	IF arrAxisCtrl[P3AxisNo.P3M1_ColdpreWhirling].Cmd.arrbRealPoint[1] AND NOT arrAxisCtrl[P3AxisNo.P3M1_ColdpreWhirling].Status.Moving THEN
		ColdpreWhirlTorMark:=FALSE;//冷压上料夹旋转力矩超限报警标志
		Init_step[1]:=170;
	END_IF	
	

	
	
170://冷压上料夹旋转在初始位且已停止，则冷压上料夹升降开始回零
INIT_TON[7].IN:=TRUE;
IF arrAxisCtrl[P3AxisNo.P3M1_ColdpreWhirling].Cmd.arrbRealPoint[1] AND NOT arrAxisCtrl[P3AxisNo.P3M1_ColdpreWhirling].Status.Moving AND  INIT_TON[7].Q THEN
	arrAxisCtrl[P3AxisNo.P3M1_ColdpreUpDown].Cmd.bHome:=TRUE;//冷压上料升降回零
	INIT_TON[7].IN:=FALSE;
	Init_step[1]:=180;
	END_IF
	

180://冷压上料夹升降回零完成
INIT_TON[9].IN:=TRUE;
	IF  arrAxisCtrl[P3AxisNo.P3M1_ColdpreUpDown].Status.Homed AND NOT arrAxisCtrl[P3AxisNo.P3M1_ColdpreUpDown].Status.Moving  AND  INIT_TON[9].Q  THEN
		Init_step[1]:=190;
		arrAxisCtrl[P3AxisNo.P3M1_ColdpreUpDown].Cmd.bHome:=FALSE;	
		INIT_TON[9].IN:=FALSE;
	END_IF

190://冷压上料夹升降到初始位
	IF  NOT arrAxisCtrl[P3AxisNo.P3M1_ColdpreUpDown].Cmd.arrbRealPoint[1] 
	AND NOT arrAxisCtrl[P3AxisNo.P3M1_ColdpreUpDown].Status.Error 
	AND arrAxisCtrl[P3AxisNo.P3M1_ColdpreUpDown].Status.Homed 
	AND arrAxisCtrl[P3AxisNo.P3M1_ColdpreUpDown].Status.Enabled 
	AND arrAxisCtrl[P3AxisNo.P3M1_ColdpreUpDown].Status.NoMoving THEN
		arrAxisCtrl[P3AxisNo.P3M1_ColdpreUpDown].Cmd.iGoSetPos:=1;	//冷压上料升降回初始位
	END_IF

	
	IF  arrAxisCtrl[P3AxisNo.P3M1_ColdpreUpDown].Cmd.arrbRealPoint[1] AND NOT arrAxisCtrl[P3AxisNo.P3M1_ColdpreUpDown].Status.Moving  THEN
		Init_step[1]:=200;
	END_IF


	
200:
Step30:=1;
Init_step[1]:=999;

999://冷压上料初始化完成
IF Init_step[1]=999 THEN
INIT_TON[20].IN:=FALSE;
LateBlanking_init_OK[1]:=TRUE;
END_IF

END_CASE
END_IF


IF 	arrAxisCtrl[P3AxisNo.P3M1_ColdpreLine].Status.Error OR arrAxisCtrl[P3AxisNo.P3M1_ColdpreUpDown].Status.Error OR
	arrAxisCtrl[P3AxisNo.P3M1_ColdpreWhirling].Status.Error OR  arrAxisCtrl[P3AxisNo.P3M1_ColdpreRetracting].Status.Error THEN
	Init_step[1]:=0;
END_IF

IF   P3_SystemRUN.btnStop OR NOT P3Button.LateStop THEN
	Init_step[1]:=0;
	Init_step[2]:=0;
	Init_step[3]:=0;
	Init_step[4]:=0;
	Init_step[5]:=0;
	Init_step[6]:=0;
	Init_step[7]:=0;
	Init_step[8]:=0;
END_IF

END_PROGRAM

// ---- P3POUs/POUs/Init/L_Init2.TcPOU
PROGRAM L_Init2
VAR
	INIT_TON  :ARRAY[1..20] OF Tc2_Standard.TON;
END_VAR

INIT_TON[1](PT:=T#2S);
INIT_TON[2](PT:=T#2S);
INIT_TON[3](PT:=T#2S);
INIT_TON[4](PT:=T#2S);
INIT_TON[5](PT:=T#2S);
INIT_TON[6](PT:=T#2S);
INIT_TON[7](PT:=T#2S);
INIT_TON[8](PT:=T#2S);
INIT_TON[9](PT:=T#2S);
INIT_TON[10](PT:=T#3S);
INIT_TON[20](PT:=T#60S);//冷压驱动回原超时计时

IF INIT_TON[20].Q THEN
	Init_step[2]:=0;
	P3_Error[121]:=TRUE;//冷压驱动回原超时报警
	INIT_TON[20].IN:=FALSE;
END_IF
//冷压托板开合回原条件
IF arrAxisCtrl[P3AxisNo.P3M1_ColdpreSupPlateLine].Status.Enabled AND NOT arrAxisCtrl[P3AxisNo.P3M1_ColdpreSupPlateLine].Status.Error AND P3_SystemRUN.iMode=3 
AND (arrAxisCtrlV2[P3AxisNo.P3_M2_OvenRetracting].Cmd.arrbRealPoint[43] OR (LREAL_TO_REAL(arrAxisCtrlV2[P3AxisNo.P3_M2_OvenCarrying].Status.fActPos)>=(arrAxisParV2[P3AxisNo.P3_M2_OvenCarrying].arrTargetPoint[1]-5)
AND  arrAxisCtrlV2[P3AxisNo.P3_M2_OvenCarrying].Status.Homed)) 
AND (arrAxisCtrl[P3AxisNo.P3M1_ColdpreRetracting].Cmd.arrbRealPoint[1] OR (LREAL_TO_REAL(arrAxisCtrl[P3AxisNo.P3M1_ColdpreLine].Status.fActPos)<=(arrAxisPar[P3AxisNo.P3M1_ColdpreLine].arrTargetPoint[2]+5)
AND  arrAxisCtrl[P3AxisNo.P3M1_ColdpreLine].Status.Homed))
AND  arrAxisCtrl[P3AxisNo.P3M1_ColdpreActuated].Cmd.arrbRealPoint[1]  THEN
   arrAxisCtrl[P3AxisNo.P3M1_ColdpreSupPlateLine].Cmd.Home_Condition:=TRUE;
   ELSE 
   arrAxisCtrl[P3AxisNo.P3M1_ColdpreSupPlateLine].Cmd.Home_Condition:=FALSE;
 END_IF

//冷压驱动回原条件
IF arrAxisCtrl[P3AxisNo.P3M1_ColdpreActuated].Status.Enabled AND NOT arrAxisCtrl[P3AxisNo.P3M1_ColdpreActuated].Status.Error AND P3_SystemRUN.iMode=3 THEN
   arrAxisCtrl[P3AxisNo.P3M1_ColdpreActuated].Cmd.Home_Condition:=TRUE;
   ELSE 
   arrAxisCtrl[P3AxisNo.P3M1_ColdpreActuated].Cmd.Home_Condition:=FALSE;
 END_IF










///////////////////////冷压初始化
IF P3_SystemRUN.iMode=3  THEN
IF LateBlanking_init_start[2]  THEN
	Init_step[2]:=1;
	LateBlanking_init_OK[2]:=FALSE;
	LateBlanking_init_start[2]:=FALSE;
END_IF
END_IF


IF P3_SystemRUN.iMode=3 AND LateBlanking_init_OK[1] AND  LateBlanking_init_OK[3] THEN
CASE Init_step[2] OF
1://冷压电芯记忆清除
	INIT_TON[20].IN:=TRUE;
	Permit_Cold_Press:=FALSE;	
	Cold_Press_Finish:=FALSE;	
	Step31:=0;
	INIT_TON[10].IN:=FALSE;
	ColdPress_start:=FALSE;
	MEMSET(ADR(CellMemory[CellNo.Coldpress]),0,SIZEOF(CellMemory[CellNo.Coldpress]));
	Init_step[2]:=10;//信号复位
	
10://冷压麦拉张紧气缸打开
arrCyCtrl[P3CYNo.P3ColdPressTensed].Cmd.bON:=TRUE;
Init_step[2]:=20;//气缸打开

20://冷压驱动停止信号复位
	arrAxisCtrl[P3AxisNo.P3M1_ColdpreActuated].Cmd.bStop:=TRUE;
	arrAxisCtrl[P3AxisNo.P3M1_ColdpreSupPlateLine].Cmd.bStop:=TRUE;//轴停止
	INIT_TON[1].IN:=TRUE;
	IF INIT_TON[1].Q THEN
		Init_step[2]:=30;
	arrAxisCtrl[P3AxisNo.P3M1_ColdpreActuated].Cmd.bStop:=FALSE;
	arrAxisCtrl[P3AxisNo.P3M1_ColdpreSupPlateLine].Cmd.bStop:=FALSE;
	INIT_TON[1].IN:=FALSE;	
	END_IF

30://冷压驱动轴复位
    arrAxisCtrl[P3AxisNo.P3M1_ColdpreActuated].Cmd.bReset:=TRUE;
	arrAxisCtrl[P3AxisNo.P3M1_ColdpreSupPlateLine].Cmd.bReset:=TRUE;//轴复位
	INIT_TON[2].IN:=TRUE;
	
	IF INIT_TON[2].Q THEN
		Init_step[2]:=40;
	    arrAxisCtrl[P3AxisNo.P3M1_ColdpreActuated].Cmd.bReset:=FALSE;
		arrAxisCtrl[P3AxisNo.P3M1_ColdpreSupPlateLine].Cmd.bReset:=FALSE;
		INIT_TON[2].IN:=FALSE;
	END_IF

40://冷压驱动、冷压托板开合轴上使能
    arrAxisCtrl[P3AxisNo.P3M1_ColdpreActuated].Cmd.bEnable:=TRUE;
	arrAxisCtrl[P3AxisNo.P3M1_ColdpreSupPlateLine].Cmd.bEnable:=TRUE;//轴上使能
	IF arrAxisCtrl[P3AxisNo.P3M1_ColdpreActuated].Status.Enabled AND arrAxisCtrl[P3AxisNo.P3M1_ColdpreSupPlateLine].Status.Enabled THEN
		Init_step[2]:=50;
	END_IF

50://冷压驱动开始回零
arrAxisCtrl[P3AxisNo.P3M1_ColdpreActuated].Cmd.bHome:=TRUE;
Init_step[2]:=60;

60://冷压驱动回零完成
INIT_TON[3].IN:=TRUE;
IF arrAxisCtrl[P3AxisNo.P3M1_ColdpreActuated].Status.Homed AND NOT arrAxisCtrl[P3AxisNo.P3M1_ColdpreActuated].Status.Moving AND INIT_TON[3].Q THEN
	Init_step[2]:=70;
    arrAxisCtrl[P3AxisNo.P3M1_ColdpreActuated].Cmd.bHome:=FALSE;
	INIT_TON[3].IN:=FALSE;
END_IF

70://冷压驱动到初始位
IF NOT arrAxisCtrl[P3AxisNo.P3M1_ColdpreActuated].Cmd.arrbRealPoint[1] AND NOT arrAxisCtrl[P3AxisNo.P3M1_ColdpreActuated].Status.Error AND arrAxisCtrl[P3AxisNo.P3M1_ColdpreActuated].Status.Homed 
	AND arrAxisCtrl[P3AxisNo.P3M1_ColdpreActuated].Status.Enabled AND arrAxisCtrl[P3AxisNo.P3M1_ColdpreActuated].Status.NoMoving THEN
	arrAxisCtrl[P3AxisNo.P3M1_ColdpreActuated].Cmd.iGoSetPos:=1;//冷压驱动回初始位	
END_IF

IF 	arrAxisCtrl[P3AxisNo.P3M1_ColdpreActuated].Cmd.arrbRealPoint[1]  AND NOT arrAxisCtrl[P3AxisNo.P3M1_ColdpreActuated].Status.Moving THEN
	Init_step[2]:=80;
END_IF


80://冷压托板开合开始回零
arrAxisCtrl[P3AxisNo.P3M1_ColdpreSupPlateLine].Cmd.bHome:=TRUE;
Init_step[2]:=90;
	
90://冷压托板开合回零完成，冷压麦拉张紧气缸打开
INIT_TON[8].IN:=TRUE;
	IF 	arrAxisCtrl[P3AxisNo.P3M1_ColdpreSupPlateLine].Status.Homed AND arrAxisCtrl[P3AxisNo.P3M1_ColdpreSupPlateLine].Status.NoMoving AND  INIT_TON[8].Q THEN
		Init_step[2]:=100;
		arrAxisCtrl[P3AxisNo.P3M1_ColdpreSupPlateLine].Cmd.bHome:=FALSE;
		arrCyCtrl[P3CYNo.P3ColdPressTensed].Cmd.bON:=TRUE;//冷压麦拉膜气缸张紧
		INIT_TON[8].IN:=FALSE;
		END_IF
100://冷压托板开合到张开位检查有无电芯
    IF  NOT arrAxisCtrl[P3AxisNo.P3M1_ColdpreSupPlateLine].Cmd.arrbRealPoint[2] AND NOT arrAxisCtrl[P3AxisNo.P3M1_ColdpreSupPlateLine].Status.Error AND arrAxisCtrl[P3AxisNo.P3M1_ColdpreSupPlateLine].Status.Homed 
		AND arrAxisCtrl[P3AxisNo.P3M1_ColdpreSupPlateLine].Status.Enabled AND arrAxisCtrl[P3AxisNo.P3M1_ColdpreSupPlateLine].Status.NoMoving THEN
		arrAxisCtrl[P3AxisNo.P3M1_ColdpreSupPlateLine].Cmd.iGoSetPos:=2;//冷压托板开合去张开位
	END_IF 
    IF arrAxisCtrl[P3AxisNo.P3M1_ColdpreSupPlateLine].Cmd.arrbRealPoint[2] 
	AND arrAxisCtrl[P3AxisNo.P3M1_ColdpreSupPlateLine].Status.NoMoving 
	AND NOT P3Senser.P3_ColdEmptyPress THEN
		Init_step[2]:=110;	
	ELSIF arrAxisCtrl[P3AxisNo.P3M1_ColdpreSupPlateLine].Cmd.arrbRealPoint[2] 
	AND arrAxisCtrl[P3AxisNo.P3M1_ColdpreSupPlateLine].Status.NoMoving 
	AND  P3Senser.P3_ColdEmptyPress THEN
		Init_step[2]:=888;	
		P3_Error[74]:=TRUE;//冷压初始化时，电芯未取走报警！
	END_IF
	
110://冷压托板开合到初始位
	IF  NOT arrAxisCtrl[P3AxisNo.P3M1_ColdpreSupPlateLine].Cmd.arrbRealPoint[1] AND NOT arrAxisCtrl[P3AxisNo.P3M1_ColdpreSupPlateLine].Status.Error AND arrAxisCtrl[P3AxisNo.P3M1_ColdpreSupPlateLine].Status.Homed 
		AND arrAxisCtrl[P3AxisNo.P3M1_ColdpreSupPlateLine].Status.Enabled AND arrAxisCtrl[P3AxisNo.P3M1_ColdpreSupPlateLine].Status.NoMoving THEN
		arrAxisCtrl[P3AxisNo.P3M1_ColdpreSupPlateLine].Cmd.iGoSetPos:=1;//冷压托板开合回初始位	
	END_IF
    IF  arrAxisCtrl[P3AxisNo.P3M1_ColdpreSupPlateLine].Cmd.arrbRealPoint[1] AND arrAxisCtrl[P3AxisNo.P3M1_ColdpreSupPlateLine].Status.NoMoving THEN
		Init_step[2]:=120;
		
	END_IF

	
120:
Step31:=1;
Init_step[2]:=999;

999://冷压回零完成
IF Init_step[2]=999 THEN
INIT_TON[20].IN:=FALSE;
LateBlanking_init_OK[2]:=TRUE;
END_IF

END_CASE
END_IF

IF arrAxisCtrl[P3AxisNo.P3M1_ColdpreSupPlateLine].Status.Error OR arrAxisCtrl[P3AxisNo.P3M1_ColdpreActuated].Status.Error THEN
	Init_step[2]:=0;
END_IF

END_PROGRAM

// ---- P3POUs/POUs/Init/L_Init3.TcPOU
PROGRAM L_Init3
VAR
	INIT_TON  :ARRAY[1..20] OF Tc2_Standard.TON;
END_VAR

INIT_TON[1](PT:=T#2S);
INIT_TON[2](PT:=T#2S);
INIT_TON[3](PT:=T#2S);
INIT_TON[4](PT:=T#2S);
INIT_TON[5](PT:=T#2S);
INIT_TON[6](PT:=T#2S);
INIT_TON[7](PT:=T#2S);
INIT_TON[8](PT:=T#2S);
INIT_TON[9](PT:=T#2S);
INIT_TON[10](PT:=T#3S);
INIT_TON[20](PT:=T#90S);//烤箱上料回原超时计时

IF INIT_TON[20].Q THEN
	Init_step[3]:=0;
	P3_Error[122]:=TRUE;//烤箱上料回原超时报警
	INIT_TON[20].IN:=FALSE;
END_IF
//烤箱上料夹搬运回原条件
IF arrAxisCtrlV2[P3AxisNo.P3_M2_OvenCarrying].Status.Enabled AND NOT arrAxisCtrlV2[P3AxisNo.P3_M2_OvenCarrying].Status.Error AND P3_SystemRUN.iMode=3 
AND arrAxisCtrlV2[P3AxisNo.P3_M2_OvenRetracting].Cmd.arrbRealPoint[43] AND Oven_CYOFF_condition THEN
   arrAxisCtrlV2[P3AxisNo.P3_M2_OvenCarrying].Cmd.Home_Condition:=TRUE;
   ELSE 
   arrAxisCtrlV2[P3AxisNo.P3_M2_OvenCarrying].Cmd.Home_Condition:=FALSE;
 END_IF

//烤箱上料夹进退回原条件
IF arrAxisCtrlV2[P3AxisNo.P3_M2_OvenRetracting].Status.Enabled AND NOT arrAxisCtrl[P3AxisNo.P3_M2_OvenRetracting].Status.Error AND P3_SystemRUN.iMode=3  THEN
   arrAxisCtrlV2[P3AxisNo.P3_M2_OvenRetracting].Cmd.Home_Condition:=TRUE;
   ELSE 
   arrAxisCtrlV2[P3AxisNo.P3_M2_OvenRetracting].Cmd.Home_Condition:=FALSE;
 END_IF

//烤箱上料夹升降回原条件
IF arrAxisCtrlV2[P3AxisNo.P3_M2_OvenUpDown].Status.Enabled AND NOT arrAxisCtrlV2[P3AxisNo.P3_M2_OvenUpDown].Status.Error AND P3_SystemRUN.iMode=3  
AND arrAxisCtrlV2[P3AxisNo.P3_M2_OvenRetracting].Cmd.arrbRealPoint[43] AND Oven_CYOFF_condition THEN
   arrAxisCtrlV2[P3AxisNo.P3_M2_OvenUpDown].Cmd.Home_Condition:=TRUE;
   ELSE 
   arrAxisCtrlV2[P3AxisNo.P3_M2_OvenUpDown].Cmd.Home_Condition:=FALSE;
 END_IF





//烤箱上下料初始化
IF P3_SystemRUN.iMode=3 THEN
IF LateBlanking_init_start[3] AND Oven_CYOFF_condition THEN
	Init_step[3]:=1;
	LateBlanking_init_OK[3]:=FALSE;
	LateBlanking_init_start[3]:=FALSE;
	ELSIF LateBlanking_init_start[3] AND NOT Oven_CYOFF_condition THEN
		Init_step[3]:=0;
		LateBlanking_init_OK[3]:=FALSE;
		LateBlanking_init_start[3]:=FALSE;
		P3_Error[28]:=TRUE;//初始化过程中，烤箱门未完成关闭，请完全关闭再重新启动烤箱初始化
END_IF
END_IF



IF P3_SystemRUN.iMode=3 THEN
CASE Init_step[3] OF

1:	//冷压下料到烤箱及烤箱下料到热压时电芯记忆清除
	INIT_TON[20].IN:=TRUE;
	Step32:=0;	
	INIT_TON[10].IN:=FALSE;
	MEMSET(ADR(CellMemory[CellNo.OvenMoveClip1]),0,SIZEOF(CellMemory[CellNo.OvenMoveClip1]));
	MEMSET(ADR(CellMemory[CellNo.OvenMoveClip2]),0,SIZEOF(CellMemory[CellNo.OvenMoveClip2]));
	Init_step[3]:=10;//信号复位
	
10://烤箱上料夹气缸关闭
arrCyCtrl[P3CYNo.P3OvenMoveClip].Cmd.bOFF:=TRUE;
IF  arrCyCtrl[P3CYNo.P3OvenMoveClip].Status.OFFState AND NOT arrCyCtrl[P3CYNo.P3OvenMoveClip].Status.Error2  THEN
	Init_step[3]:=20;
END_IF//



20://烤箱上料夹各轴停止信号复位
	arrAxisCtrlV2[P3AxisNo.P3_M2_OvenCarrying].Cmd.bStop:=TRUE;       arrAxisCtrlV2[P3AxisNo.P3_M2_OvenUpDown].Cmd.bStop:=TRUE;
	arrAxisCtrlV2[P3AxisNo.P3_M2_OvenRetracting].Cmd.bStop:=TRUE;     //轴停止
	INIT_TON[1].IN:=TRUE;
	IF INIT_TON[1].Q THEN
		Init_step[3]:=30;
		arrAxisCtrlV2[P3AxisNo.P3_M2_OvenCarrying].Cmd.bStop:=FALSE;       arrAxisCtrlV2[P3AxisNo.P3_M2_OvenUpDown].Cmd.bStop:=FALSE;
		arrAxisCtrlV2[P3AxisNo.P3_M2_OvenRetracting].Cmd.bStop:=FALSE;    
		INIT_TON[1].IN:=FALSE;	
	END_IF

30://烤箱上料夹各轴复位
	arrAxisCtrlV2[P3AxisNo.P3_M2_OvenCarrying].Cmd.bReset:=TRUE;       arrAxisCtrlV2[P3AxisNo.P3_M2_OvenUpDown].Cmd.bReset:=TRUE;
	arrAxisCtrlV2[P3AxisNo.P3_M2_OvenRetracting].Cmd.bReset:=TRUE;     //轴复位
	INIT_TON[2].IN:=TRUE;
	
	IF INIT_TON[2].Q THEN
		Init_step[3]:=40;
		arrAxisCtrlV2[P3AxisNo.P3_M2_OvenCarrying].Cmd.bReset:=FALSE;       arrAxisCtrlV2[P3AxisNo.P3_M2_OvenUpDown].Cmd.bReset:=FALSE;
		arrAxisCtrlV2[P3AxisNo.P3_M2_OvenRetracting].Cmd.bReset:=FALSE;     
		INIT_TON[2].IN:=FALSE;
	END_IF

40://烤箱上料夹各轴上使能
	arrAxisCtrlV2[P3AxisNo.P3_M2_OvenCarrying].Cmd.bEnable:=TRUE;       arrAxisCtrlV2[P3AxisNo.P3_M2_OvenUpDown].Cmd.bEnable:=TRUE;
	arrAxisCtrlV2[P3AxisNo.P3_M2_OvenRetracting].Cmd.bEnable:=TRUE;     //轴上使能
	IF  arrAxisCtrlV2[P3AxisNo.P3_M2_OvenCarrying].Status.Enabled AND arrAxisCtrlV2[P3AxisNo.P3_M2_OvenUpDown].Status.Enabled
		AND arrAxisCtrlV2[P3AxisNo.P3_M2_OvenRetracting].Status.Enabled  THEN
		Init_step[3]:=50;
	END_IF

50://烤箱上料夹进退开始回零
arrAxisCtrlV2[P3AxisNo.P3_M2_OvenRetracting].Cmd.bHome:=TRUE;//烤箱上料进退回零
Init_step[3]:=60;

60://烤箱上料夹进退回零完成
INIT_TON[4].IN:=TRUE;
IF arrAxisCtrlV2[P3AxisNo.P3_M2_OvenRetracting].Status.Homed AND NOT arrAxisCtrlV2[P3AxisNo.P3_M2_OvenRetracting].Status.Moving AND  INIT_TON[4].Q  THEN
	Init_step[3]:=70;
    arrAxisCtrlV2[P3AxisNo.P3_M2_OvenRetracting].Cmd.bHome:=FALSE;
	INIT_TON[4].IN:=FALSE;
END_IF

70://烤箱上料夹进退到初始位
IF  NOT arrAxisCtrlV2[P3AxisNo.P3_M2_OvenRetracting].Cmd.arrbRealPoint[43] AND NOT arrAxisCtrlV2[P3AxisNo.P3_M2_OvenRetracting].Status.Error AND arrAxisCtrlV2[P3AxisNo.P3_M2_OvenRetracting].Status.Homed 
	AND arrAxisCtrlV2[P3AxisNo.P3_M2_OvenRetracting].Status.Enabled AND arrAxisCtrlV2[P3AxisNo.P3_M2_OvenRetracting].Status.NoMoving THEN
	arrAxisCtrlV2[P3AxisNo.P3_M2_OvenRetracting].Cmd.iGoSetPos:=43;
	OvenRetractTorMark:=TRUE;//烤箱上料夹进退力矩超限报警标志
END_IF 

IF  arrAxisCtrlV2[P3AxisNo.P3_M2_OvenRetracting].Cmd.arrbRealPoint[43]  AND Oven_POS1  AND NOT arrAxisCtrlV2[P3AxisNo.P3_M2_OvenRetracting].Status.Moving THEN
	OvenRetractTorMark:=FALSE;//烤箱上料夹进退力矩超限报警标志
	Init_step[3]:=90;
	
END_IF



90://没有烤箱气缸报警或轴急停且烤箱全部关闭，则烤箱上料夹升降开始回零
	IF  NOT Oven_CY_STOP AND Oven_CYOFF_condition THEN
		arrAxisCtrlV2[P3AxisNo.P3_M2_OvenUpDown].Cmd.bHome:=TRUE;//烤箱上料升降回零
		Init_step[3]:=100;
	END_IF
	

100://烤箱上料夹升降回零完成
INIT_TON[9].IN:=TRUE;
	IF  arrAxisCtrlV2[P3AxisNo.P3_M2_OvenUpDown].Status.Homed AND NOT arrAxisCtrlV2[P3AxisNo.P3_M2_OvenUpDown].Status.Moving AND  INIT_TON[9].Q  THEN
		Init_step[3]:=110;
		arrAxisCtrlV2[P3AxisNo.P3_M2_OvenUpDown].Cmd.bHome:=FALSE;
		INIT_TON[9].IN:=FALSE;
	END_IF

110://烤箱上料升降到初始位
	IF  NOT arrAxisCtrlV2[P3AxisNo.P3_M2_OvenUpDown].Cmd.arrbRealPoint[43] AND NOT arrAxisCtrlV2[P3AxisNo.P3_M2_OvenUpDown].Status.Error AND arrAxisCtrlV2[P3AxisNo.P3_M2_OvenUpDown].Status.Homed 
		AND arrAxisCtrlV2[P3AxisNo.P3_M2_OvenUpDown].Status.Enabled AND arrAxisCtrlV2[P3AxisNo.P3_M2_OvenUpDown].Status.NoMoving AND NOT Oven_CY_STOP AND Oven_CYOFF_condition THEN
		arrAxisCtrlV2[P3AxisNo.P3_M2_OvenUpDown].Cmd.iGoSetPos:=43;	//烤箱上料升降回初始位
	END_IF
	
	IF   arrAxisCtrlV2[P3AxisNo.P3_M2_OvenUpDown].Cmd.arrbRealPoint[43] AND NOT arrAxisCtrlV2[P3AxisNo.P3_M2_OvenUpDown].Status.Moving THEN
		Init_step[3]:=120;
	END_IF

	
120://没有烤箱气缸报警或轴急停且烤箱全部关闭，则烤箱上料夹搬运开始回零
IF NOT Oven_CY_STOP AND Oven_CYOFF_condition THEN
arrAxisCtrlV2[P3AxisNo.P3_M2_OvenCarrying].Cmd.bHome:=TRUE;//烤箱上料搬运回零
Init_step[3]:=130;
END_IF

130://烤箱上料夹搬运回零完成
INIT_TON[5].IN:=TRUE;
IF arrAxisCtrlV2[P3AxisNo.P3_M2_OvenCarrying].Status.Homed AND NOT arrAxisCtrlV2[P3AxisNo.P3_M2_OvenCarrying].Status.Moving AND INIT_TON[5].Q THEN
	Init_step[3]:=140;
	arrAxisCtrlV2[P3AxisNo.P3_M2_OvenCarrying].Cmd.bHome:=FALSE;
	INIT_TON[5].IN:=FALSE;
END_IF

140://烤箱上料夹搬运到初始位
	IF  NOT arrAxisCtrlV2[P3AxisNo.P3_M2_OvenCarrying].Cmd.arrbRealPoint[43] AND NOT arrAxisCtrlV2[P3AxisNo.P3_M2_OvenCarrying].Status.Error AND arrAxisCtrlV2[P3AxisNo.P3_M2_OvenCarrying].Status.Homed 
		AND arrAxisCtrlV2[P3AxisNo.P3_M2_OvenCarrying].Status.Enabled AND arrAxisCtrlV2[P3AxisNo.P3_M2_OvenCarrying].Status.NoMoving AND Oven_CYOFF_condition AND NOT Oven_CY_STOP THEN
		arrAxisCtrlV2[P3AxisNo.P3_M2_OvenCarrying].Cmd.iGoSetPos:=43;//箱上料平移回初始位
		OvenCarryTorMark:=TRUE;//烤箱上料夹搬运力矩超限报警标志
	END_IF 
	IF arrAxisCtrlV2[P3AxisNo.P3_M2_OvenCarrying].Cmd.arrbRealPoint[43] AND NOT arrAxisCtrlV2[P3AxisNo.P3_M2_OvenCarrying].Status.Moving THEN
		OvenCarryTorMark:=FALSE;//烤箱上料夹搬运力矩超限报警标志
		Init_step[3]:=150;
	END_IF
	
	

	

150://烤箱门全部关闭
	arrCyCtrl[P3_Oven[1]].Cmd.bOFF:=TRUE;
	arrCyCtrl[P3_Oven[2]].Cmd.bOFF:=TRUE;
	arrCyCtrl[P3_Oven[3]].Cmd.bOFF:=TRUE;
	arrCyCtrl[P3_Oven[4]].Cmd.bOFF:=TRUE;
	arrCyCtrl[P3_Oven[5]].Cmd.bOFF:=TRUE;
	arrCyCtrl[P3_Oven[6]].Cmd.bOFF:=TRUE;
	arrCyCtrl[P3_Oven[7]].Cmd.bOFF:=TRUE;
	arrCyCtrl[P3_Oven[8]].Cmd.bOFF:=TRUE;
	arrCyCtrl[P3_Oven[9]].Cmd.bOFF:=TRUE;
	arrCyCtrl[P3_Oven[10]].Cmd.bOFF:=TRUE;
	arrCyCtrl[P3_Oven[11]].Cmd.bOFF:=TRUE;
	arrCyCtrl[P3_Oven[12]].Cmd.bOFF:=TRUE;
	arrCyCtrl[P3_Oven[13]].Cmd.bOFF:=TRUE;
	arrCyCtrl[P3_Oven[14]].Cmd.bOFF:=TRUE;
	arrCyCtrl[P3_Oven[15]].Cmd.bOFF:=TRUE;
	arrCyCtrl[P3_Oven[16]].Cmd.bOFF:=TRUE;
	arrCyCtrl[P3_Oven[17]].Cmd.bOFF:=TRUE;
	arrCyCtrl[P3_Oven[18]].Cmd.bOFF:=TRUE;
	arrCyCtrl[P3_Oven[19]].Cmd.bOFF:=TRUE;
	arrCyCtrl[P3_Oven[20]].Cmd.bOFF:=TRUE;	
	arrCyCtrl[P3_Oven[21]].Cmd.bOFF:=TRUE;
	IF Oven_CYOFF_condition THEN
		Init_step[3]:=160; 	
	END_IF	
	
160:
Step32:=1;
Init_step[3]:=999;

999://烤箱上下料初始位完成
IF Init_step[3]=999 THEN
LateBlanking_init_OK[3]:=TRUE;
INIT_TON[20].IN:=FALSE;
END_IF

END_CASE
END_IF

IF arrAxisCtrlV2[P3AxisNo.P3_M2_OvenCarrying].Status.Error OR arrAxisCtrlV2[P3AxisNo.P3_M2_OvenRetracting].Status.Error OR arrAxisCtrlV2[P3AxisNo.P3_M2_OvenUpDown].Status.Error THEN
	Init_step[3]:=0;
END_IF

END_PROGRAM

// ---- P3POUs/POUs/Init/L_Init4.TcPOU
PROGRAM L_Init4
VAR
	INIT_TON  :ARRAY[1..20] OF Tc2_Standard.TON;
END_VAR

INIT_TON[1](PT:=T#2S);
INIT_TON[2](PT:=T#2S);
INIT_TON[3](PT:=T#2S);
INIT_TON[4](PT:=T#2S);
INIT_TON[5](PT:=T#2S);
INIT_TON[6](PT:=T#2S);
INIT_TON[7](PT:=T#2S);
INIT_TON[8](PT:=T#2S);
INIT_TON[9](PT:=T#2S);
INIT_TON[10](PT:=T#3S);
INIT_TON[20](PT:=T#60S);//热压驱动回原计时超时
IF INIT_TON[20].Q THEN
	Init_step[4]:=0;
	P3_Error[123]:=TRUE;//热压驱动回原超时报警
	INIT_TON[20].IN:=FALSE;
END_IF

//热压托板开合回原条件
IF arrAxisCtrl[P3AxisNo.P3_M3_HotPressingLine].Status.Enabled AND NOT arrAxisCtrl[P3AxisNo.P3_M3_HotPressingLine].Status.Error AND P3_SystemRUN.iMode=3 
AND (arrAxisCtrlV2[P3AxisNo.P3_M2_OvenRetracting].Cmd.arrbRealPoint[43] OR (LREAL_TO_REAL(arrAxisCtrlV2[P3AxisNo.P3_M2_OvenCarrying].Status.fActPos)<=(arrAxisParV2[P3AxisNo.P3_M2_OvenCarrying].arrTargetPoint[5]+5)
AND  arrAxisCtrlV2[P3AxisNo.P3_M2_OvenCarrying].Status.Homed )) 
AND LREAL_TO_REAL(arrAxisCtrl[P3AxisNo.P3_M4_WeighLine].Status.fActPos)<=(arrAxisPar[P3AxisNo.P3_M4_WeighLine].arrTargetPoint[1]+5) 
AND   arrAxisCtrl[P3AxisNo.P3_M4_WeighLine].Status.Homed  AND arrAxisCtrl[P3AxisNo.P3_M3_HotPressingActuated].Cmd.arrbRealPoint[1] THEN
   arrAxisCtrl[P3AxisNo.P3_M3_HotPressingLine].Cmd.Home_Condition:=TRUE;
   ELSE 
   arrAxisCtrl[P3AxisNo.P3_M3_HotPressingLine].Cmd.Home_Condition:=FALSE;
 END_IF
 
//热压驱动回原条件
IF arrAxisCtrl[P3AxisNo.P3_M3_HotPressingActuated].Status.Enabled AND NOT arrAxisCtrl[P3AxisNo.P3_M3_HotPressingActuated].Status.Error AND P3_SystemRUN.iMode=3 THEN
   arrAxisCtrl[P3AxisNo.P3_M3_HotPressingActuated].Cmd.Home_Condition:=TRUE;
   ELSE 
   arrAxisCtrl[P3AxisNo.P3_M3_HotPressingActuated].Cmd.Home_Condition:=FALSE;
 END_IF










//热压初始化
IF P3_SystemRUN.iMode=3 THEN
IF LateBlanking_init_start[4]  THEN
	Init_step[4]:=1;
	LateBlanking_init_OK[4]:=FALSE;
	LateBlanking_init_start[4]:=FALSE;
END_IF
END_IF


IF P3_SystemRUN.iMode=3 AND LateBlanking_init_OK[3] AND LateBlanking_init_OK[5] THEN
CASE Init_step[4] OF
1://热压电芯记忆清除,信号复位
	INIT_TON[20].IN:=TRUE;
	Permit_Hot_Press:=FALSE;
	Hot_Press_Finish:=FALSE;
	Permit_ShortTest:=FALSE;
	ShortTest_Finish:=FALSE;
	HotPress_start:=FALSE;
	Step_Short:=0;
	Step33:=0;
	INIT_TON[10].IN:=FALSE;
	MEMSET(ADR(CellMemory[CellNo.Hotpress]),0,SIZEOF(CellMemory[CellNo.Hotpress]));
	Init_step[4]:=10;//信号复位
	
10://热压麦拉气缸张开，短路测试夹气缸关闭
arrCyCtrl[P3CYNo.P3HotPressTensed].Cmd.bON:=TRUE;
arrCyCtrl[P3CYNo.P3ShortTest].Cmd.bOFF:=TRUE;
IF arrCyCtrl[P3CYNo.P3ShortTest].Status.OFFState AND NOT arrCyCtrl[P3CYNo.P3ShortTest].Status.Error2 THEN
	Init_step[4]:=20;//气缸打开
END_IF//



20://热压驱动、托板开合轴停止信号复位
	arrAxisCtrl[P3AxisNo.P3_M3_HotPressingActuated].Cmd.bStop:=TRUE;
	arrAxisCtrl[P3AxisNo.P3_M3_HotPressingLine].Cmd.bStop:=TRUE;    //轴停止
	INIT_TON[1].IN:=TRUE;
	IF INIT_TON[1].Q THEN
		Init_step[4]:=30;
	    arrAxisCtrl[P3AxisNo.P3_M3_HotPressingActuated].Cmd.bStop:=FALSE;
		arrAxisCtrl[P3AxisNo.P3_M3_HotPressingLine].Cmd.bStop:=FALSE;    
		INIT_TON[1].IN:=FALSE;	
	END_IF

30://热压驱动、托板开合轴复位
	arrAxisCtrl[P3AxisNo.P3_M3_HotPressingActuated].Cmd.bReset:=TRUE;
	arrAxisCtrl[P3AxisNo.P3_M3_HotPressingLine].Cmd.bReset:=TRUE;    //轴复位
	INIT_TON[2].IN:=TRUE;
	IF INIT_TON[2].Q THEN
		Init_step[4]:=40;
		arrAxisCtrl[P3AxisNo.P3_M3_HotPressingActuated].Cmd.bReset:=FALSE;
		arrAxisCtrl[P3AxisNo.P3_M3_HotPressingLine].Cmd.bReset:=FALSE;    
		INIT_TON[2].IN:=FALSE;
	END_IF

40://热压驱动、托板开合轴上使能
    arrAxisCtrl[P3AxisNo.P3_M3_HotPressingActuated].Cmd.bEnable:=TRUE;
	arrAxisCtrl[P3AxisNo.P3_M3_HotPressingLine].Cmd.bEnable:=TRUE;   //轴上使能
	IF  arrAxisCtrl[P3AxisNo.P3_M3_HotPressingActuated].Status.Enabled AND arrAxisCtrl[P3AxisNo.P3_M3_HotPressingLine].Status.Enabled THEN
		Init_step[4]:=50;
	END_IF

50://热压驱动开始回零
arrAxisCtrl[P3AxisNo.P3_M3_HotPressingActuated].Cmd.bHome:=TRUE;
Init_step[4]:=60;//热压回零

60://热压驱动回零完成
INIT_TON[3].IN:=TRUE;
IF arrAxisCtrl[P3AxisNo.P3_M3_HotPressingActuated].Status.Homed AND NOT arrAxisCtrl[P3AxisNo.P3_M3_HotPressingActuated].Status.Moving AND INIT_TON[3].Q THEN
	Init_step[4]:=70;
	arrAxisCtrl[P3AxisNo.P3_M3_HotPressingActuated].Cmd.bHome:=FALSE;
	INIT_TON[3].IN:=FALSE;
END_IF

70://热压驱动到初始位

IF  NOT arrAxisCtrl[P3AxisNo.P3_M3_HotPressingActuated].Cmd.arrbRealPoint[1] AND NOT arrAxisCtrl[P3AxisNo.P3_M3_HotPressingActuated].Status.Error AND arrAxisCtrl[P3AxisNo.P3_M3_HotPressingActuated].Status.Homed 
	AND arrAxisCtrl[P3AxisNo.P3_M3_HotPressingActuated].Status.Enabled AND arrAxisCtrl[P3AxisNo.P3_M3_HotPressingActuated].Status.NoMoving THEN
	arrAxisCtrl[P3AxisNo.P3_M3_HotPressingActuated].Cmd.iGoSetPos:=1;//热压驱动回初始位	
END_IF 

IF 	arrAxisCtrl[P3AxisNo.P3_M3_HotPressingActuated].Cmd.arrbRealPoint[1] AND  NOT arrAxisCtrl[P3AxisNo.P3_M3_HotPressingActuated].Status.Moving THEN
	Init_step[4]:=80;
END_IF


80://热压托板开合开始回零
arrAxisCtrl[P3AxisNo.P3_M3_HotPressingLine].Cmd.bHome:=TRUE;//热压托板开合回零
Init_step[4]:=90;
	
90://热压托板开合回零完成，热压麦拉张紧气缸打开
INIT_TON[8].IN:=TRUE;
	IF 	arrAxisCtrl[P3AxisNo.P3_M3_HotPressingLine].Status.Homed AND arrAxisCtrl[P3AxisNo.P3_M3_HotPressingLine].Status.NoMoving AND  INIT_TON[8].Q THEN
		Init_step[4]:=100;
		arrAxisCtrl[P3AxisNo.P3_M3_HotPressingLine].Cmd.bHome:=FALSE;
		arrCyCtrl[P3CYNo.P3HotPressTensed].Cmd.bON:=TRUE;//热压麦拉膜气缸张紧
		INIT_TON[8].IN:=FALSE;
		END_IF

100://热压托板开合到张开位检查有无电芯
    IF  NOT arrAxisCtrl[P3AxisNo.P3_M3_HotPressingLine].Cmd.arrbRealPoint[2] AND NOT arrAxisCtrl[P3AxisNo.P3_M3_HotPressingLine].Status.Error AND arrAxisCtrl[P3AxisNo.P3_M3_HotPressingLine].Status.Homed 
		AND arrAxisCtrl[P3AxisNo.P3_M3_HotPressingLine].Status.Enabled AND arrAxisCtrl[P3AxisNo.P3_M3_HotPressingLine].Status.NoMoving THEN
		arrAxisCtrl[P3AxisNo.P3_M3_HotPressingLine].Cmd.iGoSetPos:=2;//热压托板开合去张开位
	END_IF 

    IF arrAxisCtrl[P3AxisNo.P3_M3_HotPressingLine].Cmd.arrbRealPoint[2] 
	AND arrAxisCtrl[P3AxisNo.P3_M3_HotPressingLine].Status.NoMoving 
	AND NOT P3Senser.P3_HotEmptyPress THEN
		Init_step[4]:=110;	
	ELSIF arrAxisCtrl[P3AxisNo.P3_M3_HotPressingLine].Cmd.arrbRealPoint[2] 
	AND arrAxisCtrl[P3AxisNo.P3_M3_HotPressingLine].Status.NoMoving 
	AND  P3Senser.P3_HotEmptyPress THEN
		Init_step[4]:=888;	
		P3_Error[75]:=TRUE;//热压初始化时，电芯未取走报警！
	END_IF

110://热压托板开合到初始位
    IF  NOT arrAxisCtrl[P3AxisNo.P3_M3_HotPressingLine].Cmd.arrbRealPoint[1] AND NOT arrAxisCtrl[P3AxisNo.P3_M3_HotPressingLine].Status.Error AND arrAxisCtrl[P3AxisNo.P3_M3_HotPressingLine].Status.Homed 
		AND arrAxisCtrl[P3AxisNo.P3_M3_HotPressingLine].Status.Enabled AND arrAxisCtrl[P3AxisNo.P3_M3_HotPressingLine].Status.NoMoving THEN
		arrAxisCtrl[P3AxisNo.P3_M3_HotPressingLine].Cmd.iGoSetPos:=1;//热压托板开合去张开位
	END_IF 
	
    IF arrAxisCtrl[P3AxisNo.P3_M3_HotPressingLine].Cmd.arrbRealPoint[1] AND arrAxisCtrl[P3AxisNo.P3_M3_HotPressingLine].Status.NoMoving THEN
		Init_step[4]:=120;	
	END_IF
	
120:
Step33:=1;
Init_step[4]:=999;

999://热压回零完成
IF Init_step[4]=999 THEN
LateBlanking_init_OK[4]:=TRUE;
INIT_TON[20].IN:=FALSE;
END_IF

END_CASE
END_IF

IF arrAxisCtrl[P3AxisNo.P3_M3_HotPressingLine].Status.Error OR arrAxisCtrl[P3AxisNo.P3_M3_HotPressingActuated].Status.Error THEN
	Init_step[4]:=0;
END_IF

END_PROGRAM

// ---- P3POUs/POUs/Init/L_Init5.TcPOU
PROGRAM L_Init5
VAR
	INIT_TON2  :ARRAY[1..20] OF Tc2_Standard.TON;
END_VAR

INIT_TON2[1](PT:=T#2S);
INIT_TON2[2](PT:=T#2S);
INIT_TON2[3](PT:=T#2S);
INIT_TON2[4](PT:=T#2S);
INIT_TON2[5](PT:=T#2S);
INIT_TON2[6](PT:=T#2S);
INIT_TON2[7](PT:=T#2S);
INIT_TON2[8](PT:=T#2S);
INIT_TON2[9](PT:=T#2S);
INIT_TON2[10](PT:=T#2S);
INIT_TON2[20](PT:=T#90S);//称重上料夹回原超时计时

IF INIT_TON2[20].Q THEN
	Init_step[5]:=0;
	P3_Error[124]:=TRUE;//称重上料夹回原超时报警
	INIT_TON2[20].IN:=FALSE;
END_IF
//称重上料夹平移回原条件
IF arrAxisCtrl[P3AxisNo.P3_M4_WeighLine].Status.Enabled AND NOT arrAxisCtrl[P3AxisNo.P3_M4_WeighLine].Status.Error AND P3_SystemRUN.iMode=3 
AND  (LREAL_TO_REAL(arrAxisCtrlV2[P3AxisNo.P3_M2_OvenCarrying].Status.fActPos)<=(arrAxisParV2[P3AxisNo.P3_M2_OvenCarrying].arrTargetPoint[5]+5))
AND arrAxisCtrlV2[P3AxisNo.P3_M2_OvenCarrying].Status.Homed 
AND (LREAL_TO_REAL(arrAxisCtrl[P3AxisNo.P3_M4_SortingoutCarrying].Status.fActPos)<=(arrAxisPar[P3AxisNo.P3_M4_SortingoutCarrying].arrTargetPoint[3]+5))
AND arrAxisCtrl[P3AxisNo.P3_M4_SortingoutCarrying].Status.Homed 
AND( arrAxisCtrl[P3AxisNo.P3_M4_WeighWhirling].Cmd.arrbRealPoint[2] 
OR arrAxisCtrl[P3AxisNo.P3_M4_WeighWhirling].Cmd.arrbRealPoint[3]
OR P3_SystemRUN.TheFirstTimebool) THEN
   arrAxisCtrl[P3AxisNo.P3_M4_WeighLine].Cmd.Home_Condition:=TRUE;
   ELSE 
   arrAxisCtrl[P3AxisNo.P3_M4_WeighLine].Cmd.Home_Condition:=FALSE;
 END_IF

 //称重上料夹升降回原条件
IF arrAxisCtrl[P3AxisNo.P3_M4_WeighUpDown].Status.Enabled AND NOT arrAxisCtrl[P3AxisNo.P3_M4_WeighUpDown].Status.Error AND P3_SystemRUN.iMode=3 
AND (arrAxisCtrl[P3AxisNo.P3_M4_WeighLine].Cmd.arrbRealPoint[1]  OR arrAxisCtrl[P3AxisNo.P3_M4_WeighLine].Cmd.arrbRealPoint[4] ) THEN
   arrAxisCtrl[P3AxisNo.P3_M4_WeighUpDown].Cmd.Home_Condition:=TRUE;
   ELSE 
   arrAxisCtrl[P3AxisNo.P3_M4_WeighUpDown].Cmd.Home_Condition:=FALSE;
 END_IF

//称重上料夹旋转回原条件
IF arrAxisCtrl[P3AxisNo.P3_M4_WeighWhirling].Status.Enabled AND NOT arrAxisCtrl[P3AxisNo.P3_M4_WeighWhirling].Status.Error AND P3_SystemRUN.iMode=3 
AND arrAxisCtrl[P3AxisNo.P3_M4_WeighLine].Cmd.arrbRealPoint[4] AND (LREAL_TO_REAL(arrAxisCtrlV2[P3AxisNo.P3_M2_OvenCarrying].Status.fActPos)<=(arrAxisParV2[P3AxisNo.P3_M2_OvenCarrying].arrTargetPoint[5]+5))//安全条件
AND arrAxisCtrlV2[P3AxisNo.P3_M2_OvenCarrying].Status.Homed THEN
   arrAxisCtrl[P3AxisNo.P3_M4_WeighWhirling].Cmd.Home_Condition:=TRUE;
   ELSE 
   arrAxisCtrl[P3AxisNo.P3_M4_WeighWhirling].Cmd.Home_Condition:=FALSE;
 END_IF







//称重上料初始化
IF P3_SystemRUN.iMode=3 THEN
IF LateBlanking_init_start[5]  THEN
	Init_step[5]:=1;
	LateBlanking_init_OK[5]:=FALSE;
	LateBlanking_init_start[5]:=FALSE;
END_IF
END_IF


IF P3_SystemRUN.iMode=3 AND LateBlanking_init_OK[3] AND LateBlanking_init_OK[6] THEN
CASE Init_step[5] OF
1://称重归正气缸张开,称重上料夹电芯记忆清除
	INIT_TON2[20].IN:=TRUE;
	Step34:=0;
	P3_Weight_gross.Init:=TRUE;
	arrCyCtrl[P3CYNo.P3WgightUP].Cmd.bOFF:=TRUE;
	MEMSET(ADR(CellMemory[CellNo.WeightClip]),0,SIZEOF(CellMemory[CellNo.WeightClip]));
	Init_step[5]:=10;//信号复位	
	
10://称重上料夹气缸打开
	arrCyCtrl[P3CYNo.P3WeightFeedingClamp].Cmd.bON:=TRUE;
	IF arrCyCtrl[P3CYNo.P3WeightFeedingClamp].Status.ONState AND NOT arrCyCtrl[P3CYNo.P3WeightFeedingClamp].Status.Error1  THEN
	   Init_step[5]:=20;
	END_IF


20:
	arrAxisCtrl[P3AxisNo.P3_M4_WeighLine].Cmd.bStop:=TRUE;         arrAxisCtrl[P3AxisNo.P3_M4_WeighUpDown].Cmd.bStop:=TRUE;
	arrAxisCtrl[P3AxisNo.P3_M4_WeighWhirling].Cmd.bStop:=TRUE;     //轴停止
	INIT_TON2[1].IN:=TRUE;
	IF INIT_TON2[1].Q THEN
		Init_step[5]:=30;
		INIT_TON2[1].IN:=FALSE;
		arrAxisCtrl[P3AxisNo.P3_M4_WeighLine].Cmd.bStop:=FALSE;         arrAxisCtrl[P3AxisNo.P3_M4_WeighUpDown].Cmd.bStop:=FALSE;
		arrAxisCtrl[P3AxisNo.P3_M4_WeighWhirling].Cmd.bStop:=FALSE;     
	END_IF

30://称重上料夹各轴复位
	arrAxisCtrl[P3AxisNo.P3_M4_WeighLine].Cmd.bReset:=TRUE;         arrAxisCtrl[P3AxisNo.P3_M4_WeighUpDown].Cmd.bReset:=TRUE;
	arrAxisCtrl[P3AxisNo.P3_M4_WeighWhirling].Cmd.bReset:=TRUE;     //轴复位
	INIT_TON2[2].IN:=TRUE;
	IF INIT_TON2[2].Q THEN
		Init_step[5]:=40;
		INIT_TON2[2].IN:=FALSE;
		arrAxisCtrl[P3AxisNo.P3_M4_WeighLine].Cmd.bReset:=FALSE;         arrAxisCtrl[P3AxisNo.P3_M4_WeighUpDown].Cmd.bReset:=FALSE;
		arrAxisCtrl[P3AxisNo.P3_M4_WeighWhirling].Cmd.bReset:=FALSE;   
	END_IF	

40://称重上料夹各轴上使能
arrAxisCtrl[P3AxisNo.P3_M4_WeighLine].Cmd.bEnable:=TRUE;         arrAxisCtrl[P3AxisNo.P3_M4_WeighUpDown].Cmd.bEnable:=TRUE;
arrAxisCtrl[P3AxisNo.P3_M4_WeighWhirling].Cmd.bEnable:=TRUE;     //轴上使能
IF arrAxisCtrl[P3AxisNo.P3_M4_WeighLine].Status.Enabled  AND arrAxisCtrl[P3AxisNo.P3_M4_WeighUpDown].Status.Enabled 
	AND arrAxisCtrl[P3AxisNo.P3_M4_WeighWhirling].Status.Enabled THEN
	Init_step[5]:=50;
END_IF


50://称重上料夹平移开始回零
IF  arrAxisCtrl[P3AxisNo.P3_M4_WeighLine].Cmd.Home_Condition THEN
arrAxisCtrl[P3AxisNo.P3_M4_WeighLine].Cmd.bHome:=TRUE;
IF NOT arrAxisCtrl[P3AxisNo.P3_M4_WeighLine].Status.Homed THEN
	Init_step[5]:=60;	
END_IF
ELSE
	P3_Error[128]:=TRUE;//称重上料夹平移回原安全条件不满足，请查看烤箱上料平移，分选夹平移，称重上料旋转是否在初始位
	Init_step[5]:=0;	
END_IF


60://称重上料夹平移回零完成
	INIT_TON2[6].IN:=TRUE;
	IF INIT_TON2[6].Q AND arrAxisCtrl[P3AxisNo.P3_M4_WeighLine].Status.Homed AND arrAxisCtrl[P3AxisNo.P3_M4_WeighLine].Status.NoMoving 	THEN
		Init_step[5]:=70;
		INIT_TON2[6].IN:=FALSE;
		arrAxisCtrl[P3AxisNo.P3_M4_WeighLine].Cmd.bHome:=FALSE;
		P3_SystemRUN.TheFirstTimebool:=FALSE;
	END_IF

	
70://称重上料夹平移到初始位
IF  NOT arrAxisCtrl[P3AxisNo.P3_M4_WeighLine].Cmd.arrbRealPoint[1] 
AND NOT arrAxisCtrl[P3AxisNo.P3_M4_WeighLine].Status.Error 
AND arrAxisCtrl[P3AxisNo.P3_M4_WeighLine].Status.Homed 
AND arrAxisCtrl[P3AxisNo.P3_M4_WeighLine].Status.Enabled 
AND arrAxisCtrl[P3AxisNo.P3_M4_WeighLine].Status.NoMoving 
//AND arrAxisCtrl[P3AxisNo.P3_M4_WeighWhirling].Io.biHomeSwitch 
THEN
	arrAxisCtrl[P3AxisNo.P3_M4_WeighLine].Cmd.iGoSetPos:=1;
	WeighLineTorMark:=TRUE;//称重上料夹平移力矩超限报警标志
END_IF 

IF arrAxisCtrl[P3AxisNo.P3_M4_WeighLine].Cmd.arrbRealPoint[1] AND arrAxisCtrl[P3AxisNo.P3_M4_WeighLine].Status.NoMoving  THEN
	WeighLineTorMark:=FALSE;//称重上料夹平移力矩超限报警标志
	Init_step[5]:=80;
END_IF	
	
	
	

80://称重上料夹升降开始回零
arrAxisCtrl[P3AxisNo.P3_M4_WeighUpDown].Cmd.bHome:=TRUE;
Init_step[5]:=90;

90://称重上料夹升降回零完成
	INIT_TON2[8].IN:=TRUE;
	IF INIT_TON2[8].Q AND arrAxisCtrl[P3AxisNo.P3_M4_WeighUpDown].Status.Homed AND arrAxisCtrl[P3AxisNo.P3_M4_WeighUpDown].Status.NoMoving 	THEN
		Init_step[5]:=100;
		INIT_TON2[8].IN:=FALSE;
		arrAxisCtrl[P3AxisNo.P3_M4_WeighUpDown].Cmd.bHome:=FALSE;
	END_IF

		
100://称重上料夹平移到避让位(旋转位）

IF  NOT arrAxisCtrl[P3AxisNo.P3_M4_WeighLine].Cmd.arrbRealPoint[4] 
	AND NOT arrAxisCtrl[P3AxisNo.P3_M4_WeighLine].Status.Error 
	AND arrAxisCtrl[P3AxisNo.P3_M4_WeighLine].Status.Homed 
	AND arrAxisCtrl[P3AxisNo.P3_M4_WeighLine].Status.Enabled 
	AND arrAxisCtrl[P3AxisNo.P3_M4_WeighLine].Status.NoMoving THEN
	arrAxisCtrl[P3AxisNo.P3_M4_WeighLine].Cmd.iGoSetPos:=4;
	WeighLineTorMark:=TRUE;//称重上料夹平移力矩超限报警标志
END_IF 

IF arrAxisCtrl[P3AxisNo.P3_M4_WeighLine].Cmd.arrbRealPoint[4] AND arrAxisCtrl[P3AxisNo.P3_M4_WeighLine].Status.NoMoving  THEN
	WeighLineTorMark:=FALSE;//称重上料夹平移力矩超限报警标志
	Init_step[5]:=110;
END_IF

110://称重上料夹旋转开始回零
IF arrAxisCtrl[P3AxisNo.P3_M4_WeighLine].Cmd.arrbRealPoint[4] AND  arrAxisCtrl[P3AxisNo.P3_M4_WeighWhirling].Cmd.Home_Condition THEN
	arrAxisCtrl[P3AxisNo.P3_M4_WeighWhirling].Cmd.bHome:=TRUE;
IF NOT arrAxisCtrl[P3AxisNo.P3_M4_WeighWhirling].Status.Homed THEN
	Init_step[5]:=120;	
END_IF
ELSE
	P3_Error[129]:=TRUE;//称重上料旋转回原安全条件不满足，请查看称重上料平移是否在旋转位或烤箱上料夹平移是否在初始位
	Init_step[5]:=0;
END_IF
120://称重上料夹旋转回零完成
	INIT_TON2[7].IN:=TRUE;
	IF INIT_TON2[7].Q AND arrAxisCtrl[P3AxisNo.P3_M4_WeighWhirling].Status.Homed AND arrAxisCtrl[P3AxisNo.P3_M4_WeighWhirling].Status.NoMoving 	THEN
		Init_step[5]:=130;
		INIT_TON2[7].IN:=FALSE;
		arrAxisCtrl[P3AxisNo.P3_M4_WeighWhirling].Cmd.bHome:=FALSE;
	END_IF


130://称重上料夹旋转到热压位
IF  NOT arrAxisCtrl[P3AxisNo.P3_M4_WeighWhirling].Cmd.arrbRealPoint[3] 
AND NOT arrAxisCtrl[P3AxisNo.P3_M4_WeighWhirling].Status.Error 
AND arrAxisCtrl[P3AxisNo.P3_M4_WeighWhirling].Status.Homed 
AND arrAxisCtrl[P3AxisNo.P3_M4_WeighWhirling].Status.Enabled 
AND arrAxisCtrl[P3AxisNo.P3_M4_WeighWhirling].Status.NoMoving THEN
	arrAxisCtrl[P3AxisNo.P3_M4_WeighWhirling].Cmd.iGoSetPos:=3;
	WeighWhirlTorMark:=TRUE;//称重上料夹旋转力矩超限报警标志
END_IF 

IF arrAxisCtrl[P3AxisNo.P3_M4_WeighWhirling].Cmd.arrbRealPoint[3] AND arrAxisCtrl[P3AxisNo.P3_M4_WeighWhirling].Status.NoMoving  THEN
	WeighWhirlTorMark:=FALSE;//称重上料夹旋转力矩超限报警标志
	Init_step[5]:=140;
END_IF




140://称重上料夹升降到初始位
IF  NOT arrAxisCtrl[P3AxisNo.P3_M4_WeighUpDown].Cmd.arrbRealPoint[1] 
AND NOT arrAxisCtrl[P3AxisNo.P3_M4_WeighUpDown].Status.Error 
AND arrAxisCtrl[P3AxisNo.P3_M4_WeighUpDown].Status.Homed 
AND arrAxisCtrl[P3AxisNo.P3_M4_WeighUpDown].Status.Enabled 
AND arrAxisCtrl[P3AxisNo.P3_M4_WeighUpDown].Status.NoMoving THEN
	arrAxisCtrl[P3AxisNo.P3_M4_WeighUpDown].Cmd.iGoSetPos:=1;
END_IF

IF arrAxisCtrl[P3AxisNo.P3_M4_WeighUpDown].Cmd.arrbRealPoint[1] AND arrAxisCtrl[P3AxisNo.P3_M4_WeighUpDown].Status.NoMoving THEN
	Init_step[5]:=150;
END_IF

150://称重上料夹平移到初始位
IF  NOT arrAxisCtrl[P3AxisNo.P3_M4_WeighLine].Cmd.arrbRealPoint[1] 
AND NOT arrAxisCtrl[P3AxisNo.P3_M4_WeighLine].Status.Error 
AND arrAxisCtrl[P3AxisNo.P3_M4_WeighLine].Status.Homed 
AND arrAxisCtrl[P3AxisNo.P3_M4_WeighLine].Status.Enabled 
AND arrAxisCtrl[P3AxisNo.P3_M4_WeighLine].Status.NoMoving THEN
	arrAxisCtrl[P3AxisNo.P3_M4_WeighLine].Cmd.iGoSetPos:=1;//称重平移电机去初始位
	WeighLineTorMark:=TRUE;//称重上料夹平移力矩超限报警标志
END_IF 

IF arrAxisCtrl[P3AxisNo.P3_M4_WeighLine].Cmd.arrbRealPoint[1] AND arrAxisCtrl[P3AxisNo.P3_M4_WeighLine].Status.NoMoving  THEN
	WeighLineTorMark:=FALSE;//称重上料夹平移力矩超限报警标志
	Init_step[5]:=160;
END_IF



160:
    Step34:=1;
	Init_step[5]:=999;
	
999://称重回零完成
IF Init_step[5]=999 THEN
LateBlanking_init_OK[5]:=TRUE;
INIT_TON2[20].IN:=FALSE;
END_IF

END_CASE
END_IF

IF arrAxisCtrl[P3AxisNo.P3_M4_WeighLine].Status.Error OR arrAxisCtrl[P3AxisNo.P3_M4_WeighUpDown].Status.Error OR arrAxisCtrl[P3AxisNo.P3_M4_WeighWhirling].Status.Error THEN
	Init_step[5]:=0;
END_IF

END_PROGRAM

// ---- P3POUs/POUs/Init/L_Init6.TcPOU
PROGRAM L_Init6
VAR
	INIT_TON2  :ARRAY[1..20] OF Tc2_Standard.TON;
END_VAR

INIT_TON2[1](PT:=T#2S);
INIT_TON2[2](PT:=T#2S);
INIT_TON2[3](PT:=T#2S);
INIT_TON2[4](PT:=T#2S);
INIT_TON2[5](PT:=T#2S);
INIT_TON2[6](PT:=T#2S);
INIT_TON2[7](PT:=T#2S);
INIT_TON2[8](PT:=T#2S);
INIT_TON2[9](PT:=T#2S);
INIT_TON2[10](PT:=T#3S);
INIT_TON2[20](PT:=T#120S);//电芯分选回原计时超时
IF INIT_TON2[20].Q THEN
	Init_step[6]:=0;
	P3_Error[125]:=TRUE;//电芯分选回原超时报警
	INIT_TON2[20].IN:=FALSE;
END_IF
//电芯分选夹搬运回原条件
IF arrAxisCtrl[P3AxisNo.P3_M4_SortingoutCarrying].Status.Enabled 
AND NOT arrAxisCtrl[P3AxisNo.P3_M4_SortingoutCarrying].Status.Error 
AND P3_SystemRUN.iMode=3 
AND arrAxisCtrl[P3AxisNo.P3_M4_SortingoutUpDown].Cmd.arrbRealPoint[1] 
AND  arrCyCtrl[P3CYNo.P3CellAdvance].Status.OFFState 
AND NOT arrCyCtrl[P3CYNo.P3CellAdvance].Status.ONState
AND  LREAL_TO_REAL(arrAxisCtrl[P3AxisNo.P3_M4_OffloadingCarrying].Status.fActPos)<=arrAxisPar[P3AxisNo.P3_M4_OffloadingCarrying].arrTargetPoint[1] THEN
   arrAxisCtrl[P3AxisNo.P3_M4_SortingoutCarrying].Cmd.Home_Condition:=TRUE;
   ELSE 
   arrAxisCtrl[P3AxisNo.P3_M4_SortingoutCarrying].Cmd.Home_Condition:=FALSE;
 END_IF

//电芯分选夹升降回原条件
IF arrAxisCtrl[P3AxisNo.P3_M4_SortingoutUpDown].Status.Enabled AND NOT arrAxisCtrl[P3AxisNo.P3_M4_SortingoutUpDown].Status.Error AND P3_SystemRUN.iMode=3 THEN
   arrAxisCtrl[P3AxisNo.P3_M4_SortingoutUpDown].Cmd.Home_Condition:=TRUE;
   ELSE 
   arrAxisCtrl[P3AxisNo.P3_M4_SortingoutUpDown].Cmd.Home_Condition:=FALSE;
 END_IF

//分选初始化
IF P3_SystemRUN.iMode=3 THEN
IF LateBlanking_init_start[6]  THEN
	Init_step[6]:=1;
	LateBlanking_init_OK[6]:=FALSE;
	LateBlanking_init_start[6]:=FALSE;
END_IF
END_IF

IF P3_SystemRUN.iMode=3 AND LateBlanking_init_OK[7]THEN
CASE Init_step[6] OF

1://信号复位，分选夹及平台电芯记忆清除
	INIT_TON2[20].IN:=TRUE;
	Cold_finish:=FALSE;
	Cold_start:=FALSE;
	PC_start:=FALSE;
	PC_finish:=FALSE;
	Permit_Weigh :=FALSE;       
	Permit_Thickness:=FALSE;    
	Weigh_Finish:=FALSE;      
	Thickness_Finish:=FALSE; 
	P3_Weight_gross.Init:=TRUE;
	Step35:=0;
	MEMSET(ADR(CellMemory[CellNo.SortClip1]),0,SIZEOF(CellMemory[CellNo.SortClip1]));
	MEMSET(ADR(CellMemory[CellNo.SortClip2]),0,SIZEOF(CellMemory[CellNo.SortClip2]));
	MEMSET(ADR(CellMemory[CellNo.Weight]),0,SIZEOF(CellMemory[CellNo.Weight]));
	MEMSET(ADR(CellMemory[CellNo.Thickness]),0,SIZEOF(CellMemory[CellNo.Thickness]));
	MEMSET(ADR(CellMemory[CellNo.BlankingPlatform]),0,SIZEOF(CellMemory[CellNo.BlankingPlatform]));
	Init_step[6]:=5;//信号复位	

5:
IF P3Senser.P3_PoleMotor2_Reach THEN
arrCyCtrl[P3CYNo.P3BoxLock1_NG].Cmd.bON:=TRUE;
END_IF
IF P3Senser.P3_PoleMotor3_Reach THEN
arrCyCtrl[P3CYNo.P3BoxLock2_NG].Cmd.bON:=TRUE;
END_IF
IF P3Senser.P3_PoleMotor4_Reach THEN
arrCyCtrl[P3CYNo.P3BoxLock3_NG].Cmd.bON:=TRUE;
END_IF

IF arrCyCtrl[P3CYNo.P3BoxLock1_NG].Status.ONState 
AND arrCyCtrl[P3CYNo.P3BoxLock2_NG].Status.ONState
AND arrCyCtrl[P3CYNo.P3BoxLock3_NG].Status.ONState THEN
		stP3NgPushMoter[2].bHome:=TRUE;
		stP3NgPushMoter[3].bHome:=TRUE;
		stP3NgPushMoter[4].bHome:=TRUE;
		Init_step[6]:=10;
END_IF
	
	
10://电芯分选夹开合、测厚台托板气缸张开，测厚压板气缸关闭,分选夹归正气缸缩回
	arrCyCtrl[P3CYNo.P3ThicknessSupport].Cmd.bOFF:=TRUE;
	arrCyCtrl[P3CYNo.P3SortClamp].Cmd.bON:=TRUE;
	arrCyCtrl[P3CYNo.P3ThicknessPressure].Cmd.bOFF:=TRUE;
	arrCyCtrl[P3CYNo.P3ThicknessMeasuringSwitch].Cmd.bON:=TRUE;//测厚台切换气缸打开
	arrCyCtrl[P3CYNo.P3SortPush].Cmd.bOFF:=TRUE;//分选夹归正气缸缩回
	IF arrCyCtrl[P3CYNo.P3SortClamp].Status.ONState AND NOT arrCyCtrl[P3CYNo.P3SortClamp].Status.Error1  
	AND arrCyCtrl[P3CYNo.P3ThicknessPressure].Status.OFFState AND NOT arrCyCtrl[P3CYNo.P3ThicknessPressure].Status.Error2 
	AND arrCyCtrl[P3CYNo.P3SortPush].Status.OFFState 
	AND arrCyCtrl[P3CYNo.P3ThicknessMeasuringSwitch].Status.ONState AND NOT arrCyCtrl[P3CYNo.P3ThicknessMeasuringSwitch].Status.Error1
	AND arrCyCtrl[P3CYNo.P3ThicknessSupport].Status.OFFState AND NOT arrCyCtrl[P3CYNo.P3ThicknessSupport].Status.Error2  THEN
	   Init_step[6]:=20;
	END_IF

20://电芯分选夹升降气缸张开
arrCyCtrl[P3CYNo.P3SortLifting].Cmd.bON:=TRUE;
IF arrCyCtrl[P3CYNo.P3SortLifting].Status.ONState AND NOT arrCyCtrl[P3CYNo.P3SortLifting].Status.Error1  THEN
 Init_step[6]:=30;
 END_IF
 
30://
arrCyCtrl[P3CYNo.P3ThicknessSupport].Cmd.bON:=TRUE;
IF arrCyCtrl[P3CYNo.P3ThicknessSupport].Status.ONState AND NOT arrCyCtrl[P3CYNo.P3ThicknessSupport].Status.Error1  THEN
 Init_step[6]:=40;
END_IF

40:
    arrAxisCtrl[P3AxisNo.P3_M4_SortingoutCarrying].Cmd.bStop:=TRUE;
	arrAxisCtrl[P3AxisNo.P3_M4_SortingoutUpDown].Cmd.bStop:=TRUE;       //轴停止
	INIT_TON2[1].IN:=TRUE;
	IF INIT_TON2[1].Q THEN
		Init_step[6]:=50;
		INIT_TON2[1].IN:=FALSE;
        arrAxisCtrl[P3AxisNo.P3_M4_SortingoutCarrying].Cmd.bStop:=FALSE;
		arrAxisCtrl[P3AxisNo.P3_M4_SortingoutUpDown].Cmd.bStop:=FALSE;       
	END_IF

50://电芯分选各轴复位
	arrAxisCtrl[P3AxisNo.P3_M4_SortingoutCarrying].Cmd.bReset:=TRUE;
	arrAxisCtrl[P3AxisNo.P3_M4_SortingoutUpDown].Cmd.bReset:=TRUE;       //轴复位
	INIT_TON2[2].IN:=TRUE;
	IF INIT_TON2[2].Q THEN
		Init_step[6]:=60;
		INIT_TON2[2].IN:=FALSE;
		arrAxisCtrl[P3AxisNo.P3_M4_SortingoutCarrying].Cmd.bReset:=FALSE;
		arrAxisCtrl[P3AxisNo.P3_M4_SortingoutUpDown].Cmd.bReset:=FALSE;     
	END_IF	

60://电芯分选各轴上使能
arrAxisCtrl[P3AxisNo.P3_M4_SortingoutCarrying].Cmd.bEnable:=TRUE;
arrAxisCtrl[P3AxisNo.P3_M4_SortingoutUpDown].Cmd.bEnable:=TRUE;       //轴上使能
IF arrAxisCtrl[P3AxisNo.P3_M4_SortingoutCarrying].Status.Enabled AND arrAxisCtrl[P3AxisNo.P3_M4_SortingoutUpDown].Status.Enabled THEN
	Init_step[6]:=70;
END_IF

70://电芯分选夹升降开始回零
arrAxisCtrl[P3AxisNo.P3_M4_SortingoutUpDown].Cmd.bHome:=TRUE;
Init_step[6]:=80;

80://电芯分选夹升降回零完成
	INIT_TON2[3].IN:=TRUE;
	IF INIT_TON2[3].Q AND arrAxisCtrl[P3AxisNo.P3_M4_SortingoutUpDown].Status.Homed AND arrAxisCtrl[P3AxisNo.P3_M4_SortingoutUpDown].Status.NoMoving THEN
		Init_step[6]:=90;
		INIT_TON2[3].IN:=FALSE;
		arrAxisCtrl[P3AxisNo.P3_M4_SortingoutUpDown].Cmd.bHome:=FALSE;
	END_IF

90://电芯分选夹升降到初始位

IF NOT arrAxisCtrl[P3AxisNo.P3_M4_SortingoutUpDown].Cmd.arrbRealPoint[1] AND NOT arrAxisCtrl[P3AxisNo.P3_M4_SortingoutUpDown].Status.Error AND arrAxisCtrl[P3AxisNo.P3_M4_SortingoutUpDown].Status.Homed 
	AND arrAxisCtrl[P3AxisNo.P3_M4_SortingoutUpDown].Status.Enabled AND arrAxisCtrl[P3AxisNo.P3_M4_SortingoutUpDown].Status.NoMoving THEN
	arrAxisCtrl[P3AxisNo.P3_M4_SortingoutUpDown].Cmd.iGoSetPos:=1;//P3_M4电芯分拣夹升降去初始位
END_IF

IF 		arrAxisCtrl[P3AxisNo.P3_M4_SortingoutUpDown].Cmd.arrbRealPoint[1] AND arrAxisCtrl[P3AxisNo.P3_M4_SortingoutUpDown].Status.NoMoving THEN
		Init_step[6]:=95;
END_IF

95://
arrCyCtrl[P3CYNo.P3CellPush].Cmd.bOFF:=TRUE;
IF arrCyCtrl[P3CYNo.P3CellPush].Status.OFFState AND NOT arrCyCtrl[P3CYNo.P3CellPush].Status.Error2 THEN
Init_step[6]:=100;	
END_IF

100://电芯分选夹旋转气缸关,电芯分选夹搬运开始回零
arrCyCtrl[P3CYNo.P3SortRotate].Cmd.bOFF:=TRUE;
arrCyCtrl[P3CYNo.P3CellAdvance].Cmd.bOFF:=TRUE;
IF arrCyCtrl[P3CYNo.P3SortRotate].Status.OFFState AND NOT arrCyCtrl[P3CYNo.P3SortRotate].Status.Error2 
AND arrCyCtrl[P3CYNo.P3CellAdvance].Status.OFFState AND NOT arrCyCtrl[P3CYNo.P3SortRotate].Status.Error2 THEN
	arrAxisCtrl[P3AxisNo.P3_M4_SortingoutCarrying].Cmd.bHome:=TRUE;
	Init_step[6]:=110;
END_IF


110://电芯分选夹搬运回零完成
	INIT_TON2[5].IN:=TRUE;
	IF INIT_TON2[5].Q AND arrAxisCtrl[P3AxisNo.P3_M4_SortingoutCarrying].Status.Homed AND arrAxisCtrl[P3AxisNo.P3_M4_SortingoutCarrying].Status.NoMoving	THEN
		Init_step[6]:=120;
		INIT_TON2[5].IN:=FALSE;
		arrAxisCtrl[P3AxisNo.P3_M4_SortingoutCarrying].Cmd.bHome:=FALSE;
	END_IF
		
120://电芯分选夹搬运到初始位
IF  NOT arrAxisCtrl[P3AxisNo.P3_M4_SortingoutCarrying].Cmd.arrbRealPoint[1] AND NOT arrAxisCtrl[P3AxisNo.P3_M4_SortingoutCarrying].Status.Error AND arrAxisCtrl[P3AxisNo.P3_M4_SortingoutCarrying].Status.Homed 
	AND arrAxisCtrl[P3AxisNo.P3_M4_SortingoutCarrying].Status.Enabled AND arrAxisCtrl[P3AxisNo.P3_M4_SortingoutCarrying].Status.NoMoving THEN
	arrAxisCtrl[P3AxisNo.P3_M4_SortingoutCarrying].Cmd.iGoSetPos:=1;//电芯分选夹搬运电机回初始位
	SortingCarryTorMark:=TRUE;//电芯分选夹搬运力矩超限报警标志
END_IF

IF 
   arrAxisCtrl[P3AxisNo.P3_M4_SortingoutCarrying].Cmd.arrbRealPoint[1] AND arrAxisCtrl[P3AxisNo.P3_M4_SortingoutCarrying].Status.NoMoving THEN
   SortingCarryTorMark:=FALSE;//电芯分选夹搬运力矩超限报警标志
	Init_step[6]:=130;
END_IF



130:
	Step35:=1;
	Thickness_Step:=1;
	Init_step[6]:=999;
	
999://电芯分选初始化完成
IF Init_step[6]=999 THEN
LateBlanking_init_OK[6]:=TRUE;
INIT_TON2[20].IN:=FALSE;
END_IF

END_CASE
END_IF

IF arrAxisCtrl[P3AxisNo.P3_M4_SortingoutCarrying].Status.Error OR arrAxisCtrl[P3AxisNo.P3_M4_SortingoutUpDown].Status.Error THEN
	Init_step[6]:=0;
END_IF

END_PROGRAM

// ---- P3POUs/POUs/Init/L_Init7.TcPOU
PROGRAM L_Init7
VAR
	INIT_TON2  :ARRAY[1..20] OF Tc2_Standard.TON;
END_VAR

INIT_TON2[1](PT:=T#2S);
INIT_TON2[2](PT:=T#2S);
INIT_TON2[3](PT:=T#2S);
INIT_TON2[4](PT:=T#2S);
INIT_TON2[5](PT:=T#2S);
INIT_TON2[6](PT:=T#2S);
INIT_TON2[7](PT:=T#2S);
INIT_TON2[8](PT:=T#2S);
INIT_TON2[9](PT:=T#2S);
INIT_TON2[10](PT:=T#2S);
INIT_TON2[20](PT:=T#60S);//电芯下料夹回原超时计时

IF INIT_TON2[20].Q THEN
	Init_step[7]:=0;
	P3_Error[126]:=TRUE;//电芯下料夹回原超时报警
	INIT_TON2[20].IN:=FALSE;
END_IF

//电芯下料夹搬运回原条件
IF arrAxisCtrl[P3AxisNo.P3_M4_OffloadingCarrying].Status.Enabled AND NOT arrAxisCtrl[P3AxisNo.P3_M4_OffloadingCarrying].Status.Error AND P3_SystemRUN.iMode=3 
AND arrAxisCtrl[P3AxisNo.P3_M4_OffloadingUpDown].Cmd.arrbRealPoint[1]  THEN
   arrAxisCtrl[P3AxisNo.P3_M4_OffloadingCarrying].Cmd.Home_Condition:=TRUE;
   ELSE 
   arrAxisCtrl[P3AxisNo.P3_M4_OffloadingCarrying].Cmd.Home_Condition:=FALSE;
 END_IF

 //电芯下料夹升降回原条件
 IF arrAxisCtrl[P3AxisNo.P3_M4_OffloadingUpDown].Status.Enabled AND NOT arrAxisCtrl[P3AxisNo.P3_M4_OffloadingUpDown].Status.Error AND P3_SystemRUN.iMode=3 THEN
   arrAxisCtrl[P3AxisNo.P3_M4_OffloadingUpDown].Cmd.Home_Condition:=TRUE;
   ELSE 
   arrAxisCtrl[P3AxisNo.P3_M4_OffloadingUpDown].Cmd.Home_Condition:=FALSE;
 END_IF




//下料初始化
IF P3_SystemRUN.iMode=3 THEN
IF LateBlanking_init_start[7]  THEN
	Init_step[7]:=1;
	LateBlanking_init_OK[7]:=FALSE;
	LateBlanking_init_start[7]:=FALSE;
END_IF	
END_IF

IF P3_SystemRUN.iMode=3 THEN
CASE Init_step[7] OF
1://信号复位，下料夹电芯记忆清除
	INIT_TON2[20].IN:=TRUE;
    Permit_BlankingRack :=FALSE; 
    Permit_TakeMaterial :=FALSE;
	Step36:=0;
	MEMSET(ADR(CellMemory[CellNo.BlankingClip]),0,SIZEOF(CellMemory[CellNo.BlankingClip]));
	Init_step[7]:=10;//信号复位	
	
10://电芯下料夹开合气缸张开
	arrCyCtrl[P3CYNo.P3BlankingClamp].Cmd.bON:=TRUE;
	IF arrCyCtrl[P3CYNo.P3BlankingClamp].Status.ONState AND NOT arrCyCtrl[P3CYNo.P3BlankingClamp].Status.Error1 THEN
	   Init_step[7]:=20;
	END_IF

20://电芯下料夹升降气缸张开
arrCyCtrl[P3CYNo.P3BlankingLifting].Cmd.bON:=TRUE;
IF arrCyCtrl[P3CYNo.P3BlankingLifting].Status.ONState AND NOT arrCyCtrl[P3CYNo.P3BlankingLifting].Status.Error1 THEN
 Init_step[7]:=30;
 END_IF
 
30:
	arrAxisCtrl[P3AxisNo.P3_M4_OffloadingCarrying].Cmd.bStop:=TRUE;
	arrAxisCtrl[P3AxisNo.P3_M4_OffloadingUpDown].Cmd.bStop:=TRUE;//轴停止
	INIT_TON2[1].IN:=TRUE;
	IF INIT_TON2[1].Q THEN
		Init_step[7]:=50;
		INIT_TON2[1].IN:=FALSE;
		arrAxisCtrl[P3AxisNo.P3_M4_OffloadingCarrying].Cmd.bStop:=FALSE;
		arrAxisCtrl[P3AxisNo.P3_M4_OffloadingUpDown].Cmd.bStop:=FALSE;
	END_IF

50://电芯下料夹各轴复位
	arrAxisCtrl[P3AxisNo.P3_M4_OffloadingCarrying].Cmd.bReset:=TRUE;
	arrAxisCtrl[P3AxisNo.P3_M4_OffloadingUpDown].Cmd.bReset:=TRUE;//轴复位
	INIT_TON2[2].IN:=TRUE;
	IF INIT_TON2[2].Q THEN
		Init_step[7]:=60;
		INIT_TON2[2].IN:=FALSE;
		arrAxisCtrl[P3AxisNo.P3_M4_OffloadingCarrying].Cmd.bReset:=FALSE;
		arrAxisCtrl[P3AxisNo.P3_M4_OffloadingUpDown].Cmd.bReset:=FALSE;
	END_IF	

60://电芯下料夹各轴使能
arrAxisCtrl[P3AxisNo.P3_M4_OffloadingCarrying].Cmd.bEnable:=TRUE;
arrAxisCtrl[P3AxisNo.P3_M4_OffloadingUpDown].Cmd.bEnable:=TRUE;//轴上使能
IF arrAxisCtrl[P3AxisNo.P3_M4_OffloadingCarrying].Status.Enabled AND arrAxisCtrl[P3AxisNo.P3_M4_OffloadingUpDown].Status.Enabled  THEN
	Init_step[7]:=70;
END_IF

70://电芯下料夹升降开始回零
arrAxisCtrl[P3AxisNo.P3_M4_OffloadingUpDown].Cmd.bHome:=TRUE;
IF NOT arrAxisCtrl[P3AxisNo.P3_M4_OffloadingUpDown].Status.Homed THEN
Init_step[7]:=80;
END_IF

80://电芯下料夹升降回零完成
	INIT_TON2[3].IN:=TRUE;
	IF INIT_TON2[3].Q AND arrAxisCtrl[P3AxisNo.P3_M4_OffloadingUpDown].Status.Homed AND arrAxisCtrl[P3AxisNo.P3_M4_OffloadingUpDown].Status.NoMoving THEN
		Init_step[7]:=90;
		INIT_TON2[3].IN:=FALSE;
		arrAxisCtrl[P3AxisNo.P3_M4_OffloadingUpDown].Cmd.bHome:=FALSE;
	END_IF

90://电芯下料夹升降电机回初始位	
IF  NOT arrAxisCtrl[P3AxisNo.P3_M4_OffloadingUpDown].Cmd.arrbRealPoint[1] AND NOT arrAxisCtrl[P3AxisNo.P3_M4_OffloadingUpDown].Status.Error AND arrAxisCtrl[P3AxisNo.P3_M4_OffloadingUpDown].Status.Homed 
	AND arrAxisCtrl[P3AxisNo.P3_M4_OffloadingUpDown].Status.Enabled AND arrAxisCtrl[P3AxisNo.P3_M4_OffloadingUpDown].Status.NoMoving THEN
	arrAxisCtrl[P3AxisNo.P3_M4_OffloadingUpDown].Cmd.iGoSetPos:=1;//电芯下料夹升降电机回初始位	
END_IF

IF 		arrAxisCtrl[P3AxisNo.P3_M4_OffloadingUpDown].Cmd.arrbRealPoint[1] AND arrAxisCtrl[P3AxisNo.P3_M4_OffloadingUpDown].Status.NoMoving THEN
		Init_step[7]:=100;
END_IF


100://电芯下料夹搬运开始回零
		arrAxisCtrl[P3AxisNo.P3_M4_OffloadingCarrying].Cmd.bHome:=TRUE;
		IF NOT arrAxisCtrl[P3AxisNo.P3_M4_OffloadingCarrying].Status.Homed  THEN
		Init_step[7]:=110;	
		END_IF
		

		
110://电芯下料夹搬运回零完成
	INIT_TON2[4].IN:=TRUE;
	IF INIT_TON2[4].Q AND arrAxisCtrl[P3AxisNo.P3_M4_OffloadingCarrying].Status.Homed AND arrAxisCtrl[P3AxisNo.P3_M4_OffloadingCarrying].Status.NoMoving THEN
		Init_step[7]:=120;
		INIT_TON2[4].IN:=FALSE;
		arrAxisCtrl[P3AxisNo.P3_M4_OffloadingCarrying].Cmd.bHome:=FALSE;
	END_IF
			
		
120://电芯下料夹搬运电机回初始位	
IF  NOT arrAxisCtrl[P3AxisNo.P3_M4_OffloadingCarrying].Cmd.arrbRealPoint[1] AND NOT arrAxisCtrl[P3AxisNo.P3_M4_OffloadingCarrying].Status.Error AND arrAxisCtrl[P3AxisNo.P3_M4_OffloadingCarrying].Status.Homed 
	AND arrAxisCtrl[P3AxisNo.P3_M4_OffloadingCarrying].Status.Enabled AND arrAxisCtrl[P3AxisNo.P3_M4_OffloadingCarrying].Status.NoMoving THEN
	arrAxisCtrl[P3AxisNo.P3_M4_OffloadingCarrying].Cmd.iGoSetPos:=1;//电芯下料夹搬运电机回初始位	
	OffloadCarryTorMark:=TRUE;//电芯下料夹搬运报警力矩设定
END_IF

IF    arrAxisCtrl[P3AxisNo.P3_M4_OffloadingCarrying].Cmd.arrbRealPoint[1] AND arrAxisCtrl[P3AxisNo.P3_M4_OffloadingCarrying].Status.NoMoving THEN
	OffloadCarryTorMark:=FALSE;//电芯下料夹搬运报警力矩设定
	Init_step[7]:=130;
END_IF

130://流水线下料旋转气缸缩回
    arrCyCtrl[P3CYNo.P3TapeSpin].Cmd.bOFF:=TRUE;
    IF arrCyCtrl[P3CYNo.P3TapeSpin].Status.OFFState THEN
       Init_step[7]:=140;			
    END_IF

140:
	Step36:=1;
	Init_step[7]:=999;
	
999://下料初始化完成
IF Init_step[7]=999 THEN
LateBlanking_init_OK[7]:=TRUE;
INIT_TON2[20].IN:=FALSE;
END_IF

END_CASE
END_IF

IF arrAxisCtrl[P3AxisNo.P3_M4_OffloadingCarrying].Status.Error OR arrAxisCtrl[P3AxisNo.P3_M4_OffloadingUpDown].Status.Error THEN
	Init_step[7]:=0;
END_IF

END_PROGRAM

// ---- P3POUs/POUs/Init/L_Init8.TcPOU
PROGRAM L_Init8
VAR
	INIT_TON2  :ARRAY[1..20] OF Tc2_Standard.TON;
END_VAR

INIT_TON2[1](PT:=T#2S);
INIT_TON2[2](PT:=T#2S);
INIT_TON2[3](PT:=T#2S);
INIT_TON2[4](PT:=T#2S);
INIT_TON2[5](PT:=T#0.2S);
INIT_TON2[6](PT:=T#2S);
INIT_TON2[7](PT:=T#2S);
INIT_TON2[20](PT:=T#60S);//热压后贴胶回原超时计时

IF INIT_TON2[20].Q THEN
	Init_step[8]:=0;
	P3_Error[127]:=TRUE;//热压后贴胶回原超时报警
	INIT_TON2[20].IN:=FALSE;
END_IF
//贴胶头回原条件
IF arrAxisCtrl[P3AxisNo.P3_TapeAdvance].Status.Enabled AND NOT arrAxisCtrl[P3AxisNo.P3_TapeAdvance].Status.Error AND P3_SystemRUN.iMode=3 
AND arrCyCtrl[P3CYNo.P3TapeLift].Status.OFFState AND NOT arrCyCtrl[P3CYNo.P3TapeLift].Status.ONState 
    AND NOT arrCyCtrl[P3CYNo.P3TapeLift].Io.DOStatus1  THEN
   arrAxisCtrl[P3AxisNo.P3_TapeAdvance].Cmd.Home_Condition:=TRUE;
   ELSE 
   arrAxisCtrl[P3AxisNo.P3_TapeAdvance].Cmd.Home_Condition:=FALSE;
 END_IF

 //贴胶平移轴回原点条件
 IF arrAxisCtrl[P3AxisNo.P3_TapeTranslation].Status.Enabled AND NOT arrAxisCtrl[P3AxisNo.P3_TapeTranslation].Status.Error AND P3_SystemRUN.iMode=3 AND
     LREAL_TO_REAL(arrAxisCtrl[P3AxisNo.P3_TapeAdvance].Status.fActPos) <= arrAxisPar[P3AxisNo.P3_TapeAdvance].arrTargetPoint[4] AND 
    ((*arrAxisCtrl[P3AxisNo.P3_M4_SortingoutUpDown].Cmd.arrbRealPoint[1] OR*) LREAL_TO_REAL(arrAxisCtrl[P3AxisNo.P3_M4_SortingoutCarrying].Status.fActPos) >= (arrAxisPar[P3AxisNo.P3_M4_SortingoutCarrying].arrTargetPoint[7]-1)) AND
    ((*arrAxisCtrl[P3AxisNo.P3_M4_OffloadingUpDown].Cmd.arrbRealPoint[1] OR*) LREAL_TO_REAL(arrAxisCtrl[P3AxisNo.P3_M4_OffloadingCarrying].Status.fActPos) <= (arrAxisPar[P3AxisNo.P3_M4_OffloadingCarrying].arrTargetPoint[3]+1)) THEN
   arrAxisCtrl[P3AxisNo.P3_TapeTranslation].Cmd.Home_Condition:=TRUE;
   ELSE 
   arrAxisCtrl[P3AxisNo.P3_TapeTranslation].Cmd.Home_Condition:=FALSE;
 END_IF

 IF P3_SystemRUN.iMode=3 THEN
  IF LateBlanking_init_start[8]   THEN
	Init_step[8]:=1;
	LateBlanking_init_OK[8]:=FALSE;
  END_IF
END_IF


IF P3_SystemRUN.iMode=3 AND LateBlanking_init_OK[6] AND LateBlanking_init_OK[7] THEN//在手动状态下
	
	CASE Init_step[8]OF

1://
		INIT_TON2[20].IN:=TRUE;
		LateBlanking_init_start[8]:=FALSE;				
		Init_step[8]:=5;

5:	//判断是否有电芯
	(*IF  P3Senser.P3_CacheSensor AND arrCyCtrl[P3CYNo.P3CellPush].Io.DIOnSwitch AND arrCyCtrl[P3CYNo.P3CellAdvance].Io.DIONSwitch THEN
		Init_step[8]:=6;
	ELSE*)
	IF NOT P3Senser.P3_CacheSensor THEN
		MEMSET(ADR(CellMemory[CellNo.BlankingPlatform]),0,SIZEOF(CellMemory[CellNo.BlankingPlatform]));
		Init_step[8]:=10;
	END_IF
		

6://有电芯的情况下，全自动初始化
        StickerStandbyDone :=FALSE;//备胶完成复位
	    stickGlueDone :=FALSE;//贴胶完成复位
	    Uppercorepermit :=FALSE;//放电芯允许复位
	    Bottomsignal :=FALSE;//贴胶下料信号复位
	    StickerDoneNo1[1]:=FALSE;//已贴胶的道数复位
        StickerDoneNo1[2]:=FALSE;//已贴胶的道数复位
        StickerDoneNo1[3]:=FALSE;//已贴胶的道数复位
		StickerDoneNo1[4]:=FALSE;//已贴胶的道数复位
		StickerDoneNo1[5]:=FALSE;//已贴胶的道数复位
		StickerDoneNo1[6]:=FALSE;//已贴胶的道数复位
        LateBlanking_init_OK[8]:=FALSE;	
		Init_step[8]:=7;
7:
	arrCyCtrl[P3CYNo.P3CellPushSpin].Cmd.bON:=TRUE;//电芯旋转定位气缸缩回
	INIT_TON2[6].IN:=FALSE;
	IF arrCyCtrl[P3CYNo.P3CellPushSpin].Status.ONState THEN	
        Init_step[8]:=8;
	END_IF	 
8:	
	arrCyCtrl[P3CYNo.P3CellSpin].Cmd.bOFF:=TRUE;//电芯旋转气缸旋转去180°
	IF NOT INIT_TON2[6].Q THEN	
		INIT_TON2[6].IN:=TRUE;
	ELSE
	   INIT_TON2[6].IN:=FALSE;
	   Init_step[8]:=9;
	END_IF	
9:
	arrCyCtrl[P3CYNo.P3CellPushSpin].Cmd.bOFF:=TRUE;//电芯旋转定位气缸伸出
	IF arrCyCtrl[P3CYNo.P3CellPushSpin].Status.OFFState AND arrCyCtrl[P3CYNo.P3CellSpin].Status.OFFState THEN	
           Init_step[8]:=10;
	END_IF		
	
	
10:	//无电芯情况下，报警人工回原电芯旋转定位气缸和电芯定位气缸
        StickerStandbyDone :=FALSE;//备胶完成复位
	    stickGlueDone :=FALSE;//贴胶完成复位
	    Uppercorepermit :=FALSE;//放电芯允许复位
	    Bottomsignal :=FALSE;//贴胶下料信号复位
	    StickerDoneNo1[1]:=FALSE;//已贴胶的道数复位
        StickerDoneNo1[2]:=FALSE;//已贴胶的道数复位
        StickerDoneNo1[3]:=FALSE;//已贴胶的道数复位
		StickerDoneNo1[4]:=FALSE;//已贴胶的道数复位
		StickerDoneNo1[5]:=FALSE;//已贴胶的道数复位
		StickerDoneNo1[6]:=FALSE;//已贴胶的道数复位
        LateBlanking_init_OK[8]:=FALSE;	
        arrCyCtrl[P3CYNo.P3CellPush].Cmd.bOFF:=	TRUE;//电芯压紧气缸缩回	
		arrCyCtrl[P3CYNo.P3TapePull].Cmd.bOFF:=TRUE;//拉胶夹紧气缸缩回
	IF  arrCyCtrl[P3CYNo.P3CellPush].Status.OFFState AND arrCyCtrl[P3CYNo.P3TapePull].Status.OFFState THEN
		Init_step[8]:=15;
	END_IF

15:
arrCyCtrl[P3CYNo.P3CellPushSpin].Cmd.bOFF:=TRUE;//电芯旋转定位气缸伸出
arrCyCtrl[P3CYNo.P3CellSpin].Cmd.bOFF:=TRUE;//电芯旋转气缸伸出
INIT_TON2[7].IN:=TRUE;
IF INIT_TON2[7].Q THEN
	IF arrCyCtrl[P3CYNo.P3CellSpin].Status.OFFState AND arrCyCtrl[P3CYNo.P3CellPushSpin].Status.OFFState THEN
		INIT_TON2[7].IN:=FALSE;
		Init_step[8]:=20;
	ELSE
		INIT_TON2[7].IN:=FALSE;
		P3_Error[49]:=TRUE;//请人工回原电芯旋转定位气缸和电芯定位气缸 
		Init_step[8]:=888;
	END_IF
END_IF			
20:			
		arrCyCtrl[P3CYNo.P3GluePush].Cmd.bOFF:=TRUE;//压胶气缸伸出
		arrCyCtrl[P3CYNo.P3TapeLift].Cmd.bOFF:=TRUE;//拉带升降气缸缩回
		arrCyCtrl[P3CYNo.P3CellAdvance].Cmd.bOFF:=TRUE;//电芯平移气缸缩回
		arrCyCtrl[P3CYNo.P3TapeBuffer].Cmd.bOFF:=TRUE;//贴胶缓存气缸缩回
		arrCyCtrl[P3CYNo.P3TapeCut].Cmd.bOFF:=TRUE;//切胶气缸缩回
		arrCyCtrl[P3CYNo.P3TapePush].Cmd.bOFF:=TRUE;//贴胶头夹紧气缸缩回
		arrCyCtrl[P3CYNo.P3TapeVacuo].Cmd.bOFF:=TRUE;//吸胶真空关闭
		
		
		IF 	arrCyCtrl[P3CYNo.P3GluePush].Status.OFFState AND  arrCyCtrl[P3CYNo.P3TapeLift].Status.OFFState AND  arrCyCtrl[P3CYNo.P3CellAdvance].Status.OFFState AND
		 arrCyCtrl[P3CYNo.P3TapeBuffer].Status.OFFState AND  arrCyCtrl[P3CYNo.P3TapeCut].Status.OFFState  AND  arrCyCtrl[P3CYNo.P3TapePush].Status.OFFState  THEN 
		Init_step[8]:=30;
		END_IF	
30:
    arrAxisCtrl[P3AxisNo.P3_TapeAdvance].Cmd.bStop:=TRUE;
	arrAxisCtrl[P3AxisNo.P3_TapeTranslation].Cmd.bStop:=TRUE;//轴停止
	INIT_TON2[1].IN:=TRUE;
	IF INIT_TON2[1].Q THEN
		INIT_TON2[1].IN:=FALSE;
		arrAxisCtrl[P3AxisNo.P3_TapeAdvance].Cmd.bStop:=FALSE;
		arrAxisCtrl[P3AxisNo.P3_TapeTranslation].Cmd.bStop:=FALSE;
		Init_step[8]:=40;
	END_IF

40:
	arrAxisCtrl[P3AxisNo.P3_TapeAdvance].Cmd.bReset:=TRUE;
	arrAxisCtrl[P3AxisNo.P3_TapeTranslation].Cmd.bReset:=TRUE;//轴复位
	INIT_TON2[2].IN:=TRUE;
	IF INIT_TON2[2].Q THEN
		INIT_TON2[2].IN:=FALSE;
		arrAxisCtrl[P3AxisNo.P3_TapeAdvance].Cmd.bReset:=FALSE;
		arrAxisCtrl[P3AxisNo.P3_TapeTranslation].Cmd.bReset:=FALSE;
		Init_step[8]:=50;
	END_IF	

50:
    arrAxisCtrl[P3AxisNo.P3_TapeAdvance].Cmd.bEnable:=TRUE;
    arrAxisCtrl[P3AxisNo.P3_TapeTranslation].Cmd.bEnable:=TRUE;//轴上使能
    IF arrAxisCtrl[P3AxisNo.P3_TapeAdvance].Status.Enabled AND arrAxisCtrl[P3AxisNo.P3_TapeTranslation].Status.Enabled  THEN
	    Init_step[8]:=60;
    END_IF	
					
60://贴胶头进退轴回原点
	IF NOT arrCyCtrl[P3CYNo.P3TapeLift].Status.ONState AND arrCyCtrl[P3CYNo.P3TapeLift].Status.OFFState 
       AND NOT arrCyCtrl[P3CYNo.P3TapeLift].Io.DOStatus1 THEN
		arrAxisCtrl[P3AxisNo.P3_TapeAdvance].Cmd.bHome:=TRUE;
		Init_step[8]:=70;
	END_IF		
70:	//贴胶头进退回零完成
		INIT_TON2[3].IN:=TRUE;				
		IF INIT_TON2[3].Q AND arrAxisCtrl[P3AxisNo.P3_TapeAdvance].Status.Homed AND arrAxisCtrl[P3AxisNo.P3_TapeAdvance].Status.NoMoving THEN 
			arrAxisCtrl[P3AxisNo.P3_TapeAdvance].Cmd.bHome:=FALSE;
			INIT_TON2[3].IN:=FALSE;
			Init_step[8]:=80;
		END_IF	
80:		
	//贴胶平移轴回原点	
	 IF  arrAxisCtrl[P3AxisNo.P3_TapeTranslation].Cmd.Home_Condition THEN	
		arrAxisCtrl[P3AxisNo.P3_TapeTranslation].Cmd.bHome:=TRUE;
		Init_step[8]:=90;	
	 END_IF		
90:		//贴胶平移开始回零
        INIT_TON2[4].IN:=TRUE;						
		IF INIT_TON2[4].Q AND arrAxisCtrl[P3AxisNo.P3_TapeTranslation].Status.Homed  AND arrAxisCtrl[P3AxisNo.P3_TapeTranslation].Status.NoMoving THEN 
			arrAxisCtrl[P3AxisNo.P3_TapeTranslation].Cmd.bHome:=FALSE;
			INIT_TON2[4].IN:=FALSE;
			Init_step[8]:=100;
		END_IF			
			
100://1=贴胶头进退轴回初始位，2=贴胶平移轴回初始位
         INIT_TON2[5].IN:=TRUE;	
		IF NOT arrAxisCtrl[P3AxisNo.P3_TapeAdvance].Cmd.arrbRealPoint[1] AND NOT  arrAxisCtrl[P3AxisNo.P3_TapeAdvance].Status.Error AND
           arrAxisCtrl[P3AxisNo.P3_TapeAdvance].Status.NoMoving AND INIT_TON2[5].Q  THEN
			arrAxisCtrl[P3AxisNo.P3_TapeAdvance].Cmd.iGoSetPos :=1;
		END_IF	
		IF NOT arrAxisCtrl[P3AxisNo.P3_TapeTranslation].Cmd.arrbRealPoint[8] AND INIT_TON2[5].Q THEN
			arrAxisCtrl[P3AxisNo.P3_TapeTranslation].Cmd.iGoSetPos :=8;
		END_IF	
		IF arrAxisCtrl[P3AxisNo.P3_TapeAdvance].Cmd.arrbRealPoint[1] AND arrAxisCtrl[P3AxisNo.P3_TapeTranslation].Cmd.arrbRealPoint[8]  THEN
			Init_step[8]:=110;
			INIT_TON2[5].IN:=FALSE;	
		END_IF
110:		
		Step37:=0;
		Step38:=1;
		Init_step[8]:=999;
999://后段贴胶回零完成
		LateBlanking_init_OK[8]:=TRUE;
		INIT_TON2[20].IN:=FALSE;		
		
END_CASE	
END_IF

END_PROGRAM

// ---- P3POUs/POUs/Auxiliary/LateBlanking_Temperature.TcPOU
PROGRAM LateBlanking_Temperature
VAR
	P3_FB_Temperature: ARRAY[1..104] OF FB_Temperature;
	i:INT;
END_VAR

ACT2();

IF Tem_HOT THEN
arrTempCtrl[1].Out.PIDRun:=TRUE;
arrTempCtrl[2].Out.PIDRun:=TRUE;
arrTempCtrl[3].Out.PIDRun:=TRUE;
arrTempCtrl[4].Out.PIDRun:=TRUE;
arrTempCtrl[5].Out.PIDRun:=TRUE;
arrTempCtrl[6].Out.PIDRun:=TRUE;
arrTempCtrl[7].Out.PIDRun:=TRUE;
arrTempCtrl[8].Out.PIDRun:=TRUE;
arrTempCtrl[9].Out.PIDRun:=TRUE;
arrTempCtrl[10].Out.PIDRun:=TRUE;
arrTempCtrl[11].Out.PIDRun:=TRUE;
arrTempCtrl[12].Out.PIDRun:=TRUE;
arrTempCtrl[13].Out.PIDRun:=TRUE;
arrTempCtrl[14].Out.PIDRun:=TRUE;
arrTempCtrl[15].Out.PIDRun:=TRUE;
arrTempCtrl[16].Out.PIDRun:=TRUE;
arrTempCtrl[17].Out.PIDRun:=TRUE;
arrTempCtrl[18].Out.PIDRun:=TRUE;
arrTempCtrl[19].Out.PIDRun:=TRUE;
arrTempCtrl[20].Out.PIDRun:=TRUE;
arrTempCtrl[21].Out.PIDRun:=TRUE;
arrTempCtrl[22].Out.PIDRun:=TRUE;
arrTempCtrl[23].Out.PIDRun:=TRUE;
arrTempCtrl[24].Out.PIDRun:=TRUE;
arrTempCtrl[25].Out.PIDRun:=TRUE;
arrTempCtrl[26].Out.PIDRun:=TRUE;
arrTempCtrl[27].Out.PIDRun:=TRUE;
arrTempCtrl[28].Out.PIDRun:=TRUE;
//arrTempCtrl[29].Out.PIDRun:=TRUE;
//arrTempCtrl[30].Out.PIDRun:=TRUE;
//arrTempCtrl[31].Out.PIDRun:=TRUE;
//arrTempCtrl[32].Out.PIDRun:=TRUE;
arrTempCtrl[33].Out.PIDRun:=TRUE;
arrTempCtrl[34].Out.PIDRun:=TRUE;
arrTempCtrl[35].Out.PIDRun:=TRUE;
arrTempCtrl[36].Out.PIDRun:=TRUE;
arrTempCtrl[37].Out.PIDRun:=TRUE;
arrTempCtrl[38].Out.PIDRun:=TRUE;
arrTempCtrl[39].Out.PIDRun:=TRUE;
arrTempCtrl[40].Out.PIDRun:=TRUE;
arrTempCtrl[41].Out.PIDRun:=TRUE;
arrTempCtrl[42].Out.PIDRun:=TRUE;
arrTempCtrl[43].Out.PIDRun:=TRUE;
arrTempCtrl[44].Out.PIDRun:=TRUE;
arrTempCtrl[45].Out.PIDRun:=TRUE;
arrTempCtrl[46].Out.PIDRun:=TRUE;
arrTempCtrl[47].Out.PIDRun:=TRUE;
arrTempCtrl[48].Out.PIDRun:=TRUE;
arrTempCtrl[49].Out.PIDRun:=TRUE;
arrTempCtrl[50].Out.PIDRun:=TRUE;
arrTempCtrl[51].Out.PIDRun:=TRUE;
arrTempCtrl[52].Out.PIDRun:=TRUE;
arrTempCtrl[53].Out.PIDRun:=TRUE;
arrTempCtrl[54].Out.PIDRun:=TRUE;
arrTempCtrl[55].Out.PIDRun:=TRUE;
arrTempCtrl[56].Out.PIDRun:=TRUE;
arrTempCtrl[57].Out.PIDRun:=TRUE;
arrTempCtrl[58].Out.PIDRun:=TRUE;
arrTempCtrl[59].Out.PIDRun:=TRUE;
arrTempCtrl[60].Out.PIDRun:=TRUE;
//arrTempCtrl[61].Out.PIDRun:=TRUE;
//arrTempCtrl[62].Out.PIDRun:=TRUE;
//arrTempCtrl[63].Out.PIDRun:=TRUE;
//arrTempCtrl[64].Out.PIDRun:=TRUE;
arrTempCtrl[65].Out.PIDRun:=TRUE;
arrTempCtrl[66].Out.PIDRun:=TRUE;
arrTempCtrl[67].Out.PIDRun:=TRUE;
arrTempCtrl[68].Out.PIDRun:=TRUE;
arrTempCtrl[69].Out.PIDRun:=TRUE;
arrTempCtrl[70].Out.PIDRun:=TRUE;
arrTempCtrl[71].Out.PIDRun:=TRUE;
arrTempCtrl[72].Out.PIDRun:=TRUE;
arrTempCtrl[73].Out.PIDRun:=TRUE;
arrTempCtrl[74].Out.PIDRun:=TRUE;
arrTempCtrl[75].Out.PIDRun:=TRUE;
arrTempCtrl[76].Out.PIDRun:=TRUE;
arrTempCtrl[77].Out.PIDRun:=TRUE;
arrTempCtrl[78].Out.PIDRun:=TRUE;
arrTempCtrl[79].Out.PIDRun:=TRUE;
arrTempCtrl[80].Out.PIDRun:=TRUE;
arrTempCtrl[81].Out.PIDRun:=TRUE;
arrTempCtrl[82].Out.PIDRun:=TRUE;
arrTempCtrl[83].Out.PIDRun:=TRUE;
arrTempCtrl[84].Out.PIDRun:=TRUE;
arrTempCtrl[85].Out.PIDRun:=TRUE;
arrTempCtrl[86].Out.PIDRun:=TRUE;
arrTempCtrl[87].Out.PIDRun:=TRUE;
arrTempCtrl[88].Out.PIDRun:=TRUE;
arrTempCtrl[89].Out.PIDRun:=TRUE;
arrTempCtrl[90].Out.PIDRun:=TRUE;
arrTempCtrl[91].Out.PIDRun:=TRUE;
arrTempCtrl[92].Out.PIDRun:=TRUE;
arrTempCtrl[93].Out.PIDRun:=TRUE;
arrTempCtrl[94].Out.PIDRun:=TRUE;
END_IF

IF Tem_Cold THEN
arrTempCtrl[1].Out.PIDRun:=FALSE;
arrTempCtrl[2].Out.PIDRun:=FALSE;
arrTempCtrl[3].Out.PIDRun:=FALSE;
arrTempCtrl[4].Out.PIDRun:=FALSE;
arrTempCtrl[5].Out.PIDRun:=FALSE;
arrTempCtrl[6].Out.PIDRun:=FALSE;
arrTempCtrl[7].Out.PIDRun:=FALSE;
arrTempCtrl[8].Out.PIDRun:=FALSE;
arrTempCtrl[9].Out.PIDRun:=FALSE;
arrTempCtrl[10].Out.PIDRun:=FALSE;
arrTempCtrl[11].Out.PIDRun:=FALSE;
arrTempCtrl[12].Out.PIDRun:=FALSE;
arrTempCtrl[13].Out.PIDRun:=FALSE;
arrTempCtrl[14].Out.PIDRun:=FALSE;
arrTempCtrl[15].Out.PIDRun:=FALSE;
arrTempCtrl[16].Out.PIDRun:=FALSE;
arrTempCtrl[17].Out.PIDRun:=FALSE;
arrTempCtrl[18].Out.PIDRun:=FALSE;
arrTempCtrl[19].Out.PIDRun:=FALSE;
arrTempCtrl[20].Out.PIDRun:=FALSE;
arrTempCtrl[21].Out.PIDRun:=FALSE;
arrTempCtrl[22].Out.PIDRun:=FALSE;
arrTempCtrl[23].Out.PIDRun:=FALSE;
arrTempCtrl[24].Out.PIDRun:=FALSE;
arrTempCtrl[25].Out.PIDRun:=FALSE;
arrTempCtrl[26].Out.PIDRun:=FALSE;
arrTempCtrl[27].Out.PIDRun:=FALSE;
arrTempCtrl[28].Out.PIDRun:=FALSE;
//arrTempCtrl[29].Out.PIDRun:=FALSE;
//arrTempCtrl[30].Out.PIDRun:=FALSE;
//arrTempCtrl[31].Out.PIDRun:=FALSE;
//arrTempCtrl[32].Out.PIDRun:=FALSE;
arrTempCtrl[33].Out.PIDRun:=FALSE;
arrTempCtrl[34].Out.PIDRun:=FALSE;
arrTempCtrl[35].Out.PIDRun:=FALSE;
arrTempCtrl[36].Out.PIDRun:=FALSE;
arrTempCtrl[37].Out.PIDRun:=FALSE;
arrTempCtrl[38].Out.PIDRun:=FALSE;
arrTempCtrl[39].Out.PIDRun:=FALSE;
arrTempCtrl[40].Out.PIDRun:=FALSE;
arrTempCtrl[41].Out.PIDRun:=FALSE;
arrTempCtrl[42].Out.PIDRun:=FALSE;
arrTempCtrl[43].Out.PIDRun:=FALSE;
arrTempCtrl[44].Out.PIDRun:=FALSE;
arrTempCtrl[45].Out.PIDRun:=FALSE;
arrTempCtrl[46].Out.PIDRun:=FALSE;
arrTempCtrl[47].Out.PIDRun:=FALSE;
arrTempCtrl[48].Out.PIDRun:=FALSE;
arrTempCtrl[49].Out.PIDRun:=FALSE;
arrTempCtrl[50].Out.PIDRun:=FALSE;
arrTempCtrl[51].Out.PIDRun:=FALSE;
arrTempCtrl[52].Out.PIDRun:=FALSE;
arrTempCtrl[53].Out.PIDRun:=FALSE;
arrTempCtrl[54].Out.PIDRun:=FALSE;
arrTempCtrl[55].Out.PIDRun:=FALSE;
arrTempCtrl[56].Out.PIDRun:=FALSE;
arrTempCtrl[57].Out.PIDRun:=FALSE;
arrTempCtrl[58].Out.PIDRun:=FALSE;
arrTempCtrl[59].Out.PIDRun:=FALSE;
arrTempCtrl[60].Out.PIDRun:=FALSE;
//arrTempCtrl[61].Out.PIDRun:=FALSE;
//arrTempCtrl[62].Out.PIDRun:=FALSE;
//arrTempCtrl[63].Out.PIDRun:=FALSE;
//arrTempCtrl[64].Out.PIDRun:=FALSE;
arrTempCtrl[65].Out.PIDRun:=FALSE;
arrTempCtrl[66].Out.PIDRun:=FALSE;
arrTempCtrl[67].Out.PIDRun:=FALSE;
arrTempCtrl[68].Out.PIDRun:=FALSE;
arrTempCtrl[69].Out.PIDRun:=FALSE;
arrTempCtrl[70].Out.PIDRun:=FALSE;
arrTempCtrl[71].Out.PIDRun:=FALSE;
arrTempCtrl[72].Out.PIDRun:=FALSE;
arrTempCtrl[73].Out.PIDRun:=FALSE;
arrTempCtrl[74].Out.PIDRun:=FALSE;
arrTempCtrl[75].Out.PIDRun:=FALSE;
arrTempCtrl[76].Out.PIDRun:=FALSE;
arrTempCtrl[77].Out.PIDRun:=FALSE;
arrTempCtrl[78].Out.PIDRun:=FALSE;
arrTempCtrl[79].Out.PIDRun:=FALSE;
arrTempCtrl[80].Out.PIDRun:=FALSE;
arrTempCtrl[81].Out.PIDRun:=FALSE;
arrTempCtrl[82].Out.PIDRun:=FALSE;
arrTempCtrl[83].Out.PIDRun:=FALSE;
arrTempCtrl[84].Out.PIDRun:=FALSE;
arrTempCtrl[85].Out.PIDRun:=FALSE;
arrTempCtrl[86].Out.PIDRun:=FALSE;
arrTempCtrl[87].Out.PIDRun:=FALSE;
arrTempCtrl[88].Out.PIDRun:=FALSE;
arrTempCtrl[89].Out.PIDRun:=FALSE;
arrTempCtrl[90].Out.PIDRun:=FALSE;
arrTempCtrl[91].Out.PIDRun:=FALSE;
arrTempCtrl[92].Out.PIDRun:=FALSE;
arrTempCtrl[93].Out.PIDRun:=FALSE;
arrTempCtrl[94].Out.PIDRun:=FALSE;
	
END_IF



//1号烤箱
IF (arrTempCtrl[1].Tem_fPV>(arrTempPar[1].fTempSet+ABS(arrTempPar[1].fTempArea)) OR arrTempCtrl[1].Tem_fPV<(arrTempPar[1].fTempSet-ABS(arrTempPar[1].fTempArea))) AND NOT P3User2_Par.Oven_Shield[1] AND P3_SystemRUN.iMode=1  THEN
	P3_Tem_Error[1]:=TRUE;//烤箱1的1板温度不在正常设定温度范围内报警
END_IF

IF (arrTempCtrl[2].Tem_fPV>(arrTempPar[2].fTempSet+ABS(arrTempPar[2].fTempArea)) OR arrTempCtrl[2].Tem_fPV<(arrTempPar[2].fTempSet-ABS(arrTempPar[2].fTempArea))) AND NOT P3User2_Par.Oven_Shield[1] AND P3_SystemRUN.iMode=1 THEN
	P3_Tem_Error[2]:=TRUE;//烤箱1的2板温度不在正常设定温度范围内报警
END_IF

IF (arrTempCtrl[3].Tem_fPV>(arrTempPar[3].fTempSet+ABS(arrTempPar[3].fTempArea)) OR arrTempCtrl[3].Tem_fPV<(arrTempPar[3].fTempSet-ABS(arrTempPar[3].fTempArea))) AND NOT P3User2_Par.Oven_Shield[1] AND P3_SystemRUN.iMode=1  THEN
	P3_Tem_Error[3]:=TRUE;//烤箱1的3板温度不在正常设定温度范围内报警
END_IF

IF (arrTempCtrl[4].Tem_fPV>(arrTempPar[4].fTempSet+ABS(arrTempPar[4].fTempArea)) OR arrTempCtrl[4].Tem_fPV<(arrTempPar[4].fTempSet-ABS(arrTempPar[4].fTempArea))) AND NOT P3User2_Par.Oven_Shield[1] AND P3_SystemRUN.iMode=1 THEN
	P3_Tem_Error[4]:=TRUE;//烤箱1的4板温度不在正常设定温度范围内报警
END_IF

//2号烤箱
IF (arrTempCtrl[5].Tem_fPV>(arrTempPar[5].fTempSet+ABS(arrTempPar[5].fTempArea)) OR arrTempCtrl[5].Tem_fPV<(arrTempPar[5].fTempSet-ABS(arrTempPar[5].fTempArea))) AND NOT P3User2_Par.Oven_Shield[4] AND P3_SystemRUN.iMode=1  THEN
	P3_Tem_Error[5]:=TRUE;//烤箱2的1板温度不在正常设定温度范围内报警
END_IF

IF (arrTempCtrl[6].Tem_fPV>(arrTempPar[6].fTempSet+ABS(arrTempPar[6].fTempArea)) OR arrTempCtrl[6].Tem_fPV<(arrTempPar[6].fTempSet-ABS(arrTempPar[6].fTempArea))) AND NOT P3User2_Par.Oven_Shield[4] AND P3_SystemRUN.iMode=1 THEN
	P3_Tem_Error[6]:=TRUE;//烤箱2的2板温度不在正常设定温度范围内报警
END_IF

IF (arrTempCtrl[7].Tem_fPV>(arrTempPar[7].fTempSet+ABS(arrTempPar[7].fTempArea)) OR arrTempCtrl[7].Tem_fPV<(arrTempPar[7].fTempSet-ABS(arrTempPar[7].fTempArea))) AND NOT P3User2_Par.Oven_Shield[4] AND P3_SystemRUN.iMode=1  THEN
	P3_Tem_Error[7]:=TRUE;//烤箱2的3板温度不在正常设定温度范围内报警
END_IF

IF (arrTempCtrl[8].Tem_fPV>(arrTempPar[8].fTempSet+ABS(arrTempPar[8].fTempArea)) OR arrTempCtrl[8].Tem_fPV<(arrTempPar[8].fTempSet-ABS(arrTempPar[8].fTempArea))) AND NOT P3User2_Par.Oven_Shield[4] AND P3_SystemRUN.iMode=1 THEN
	P3_Tem_Error[8]:=TRUE;//烤箱2的4板温度不在正常设定温度范围内报警
END_IF

//3号烤箱
IF (arrTempCtrl[9].Tem_fPV>(arrTempPar[9].fTempSet+ABS(arrTempPar[9].fTempArea)) OR arrTempCtrl[9].Tem_fPV<(arrTempPar[9].fTempSet-ABS(arrTempPar[9].fTempArea))) AND NOT P3User2_Par.Oven_Shield[7] AND P3_SystemRUN.iMode=1  THEN
	P3_Tem_Error[9]:=TRUE;//烤箱3的1板温度不在正常设定温度范围内报警
END_IF

IF (arrTempCtrl[10].Tem_fPV>(arrTempPar[10].fTempSet+ABS(arrTempPar[10].fTempArea)) OR arrTempCtrl[10].Tem_fPV<(arrTempPar[10].fTempSet-ABS(arrTempPar[10].fTempArea))) AND NOT P3User2_Par.Oven_Shield[7] AND P3_SystemRUN.iMode=1 THEN
	P3_Tem_Error[10]:=TRUE;//烤箱3的2板温度不在正常设定温度范围内报警
END_IF

IF (arrTempCtrl[11].Tem_fPV>(arrTempPar[11].fTempSet+ABS(arrTempPar[11].fTempArea)) OR arrTempCtrl[11].Tem_fPV<(arrTempPar[11].fTempSet-ABS(arrTempPar[11].fTempArea))) AND NOT P3User2_Par.Oven_Shield[7] AND P3_SystemRUN.iMode=1  THEN
	P3_Tem_Error[11]:=TRUE;//烤箱3的3板温度不在正常设定温度范围内报警
END_IF

IF (arrTempCtrl[12].Tem_fPV>(arrTempPar[12].fTempSet+ABS(arrTempPar[12].fTempArea)) OR arrTempCtrl[12].Tem_fPV<(arrTempPar[12].fTempSet-ABS(arrTempPar[12].fTempArea))) AND NOT P3User2_Par.Oven_Shield[7] AND P3_SystemRUN.iMode=1 THEN
	P3_Tem_Error[12]:=TRUE;//烤箱3的4板温度不在正常设定温度范围内报警
END_IF

//4号烤箱
IF (arrTempCtrl[13].Tem_fPV>(arrTempPar[13].fTempSet+ABS(arrTempPar[13].fTempArea)) OR arrTempCtrl[13].Tem_fPV<(arrTempPar[13].fTempSet-ABS(arrTempPar[13].fTempArea))) AND NOT P3User2_Par.Oven_Shield[10] AND P3_SystemRUN.iMode=1  THEN
	P3_Tem_Error[13]:=TRUE;//烤箱4的1板温度不在正常设定温度范围内报警
END_IF

IF (arrTempCtrl[14].Tem_fPV>(arrTempPar[14].fTempSet+ABS(arrTempPar[14].fTempArea)) OR arrTempCtrl[14].Tem_fPV<(arrTempPar[14].fTempSet-ABS(arrTempPar[14].fTempArea))) AND NOT P3User2_Par.Oven_Shield[10] AND P3_SystemRUN.iMode=1 THEN
	P3_Tem_Error[14]:=TRUE;//烤箱4的2板温度不在正常设定温度范围内报警
END_IF

IF (arrTempCtrl[15].Tem_fPV>(arrTempPar[15].fTempSet+ABS(arrTempPar[15].fTempArea)) OR arrTempCtrl[15].Tem_fPV<(arrTempPar[15].fTempSet-ABS(arrTempPar[15].fTempArea))) AND NOT P3User2_Par.Oven_Shield[10] AND P3_SystemRUN.iMode=1  THEN
	P3_Tem_Error[15]:=TRUE;//烤箱4的3板温度不在正常设定温度范围内报警
END_IF

IF (arrTempCtrl[16].Tem_fPV>(arrTempPar[16].fTempSet+ABS(arrTempPar[16].fTempArea)) OR arrTempCtrl[16].Tem_fPV<(arrTempPar[16].fTempSet-ABS(arrTempPar[16].fTempArea))) AND NOT P3User2_Par.Oven_Shield[10] AND P3_SystemRUN.iMode=1 THEN
	P3_Tem_Error[16]:=TRUE;//烤箱4的4板温度不在正常设定温度范围内报警
END_IF

//5号烤箱
IF (arrTempCtrl[17].Tem_fPV>(arrTempPar[17].fTempSet+ABS(arrTempPar[17].fTempArea)) OR arrTempCtrl[17].Tem_fPV<(arrTempPar[17].fTempSet-ABS(arrTempPar[17].fTempArea))) AND NOT P3User2_Par.Oven_Shield[13] AND P3_SystemRUN.iMode=1  THEN
	P3_Tem_Error[17]:=TRUE;//烤箱5的1板温度不在正常设定温度范围内报警
END_IF

IF (arrTempCtrl[18].Tem_fPV>(arrTempPar[18].fTempSet+ABS(arrTempPar[18].fTempArea)) OR arrTempCtrl[18].Tem_fPV<(arrTempPar[18].fTempSet-ABS(arrTempPar[18].fTempArea))) AND NOT P3User2_Par.Oven_Shield[13] AND P3_SystemRUN.iMode=1 THEN
	P3_Tem_Error[18]:=TRUE;//烤箱5的2板温度不在正常设定温度范围内报警
END_IF

IF (arrTempCtrl[19].Tem_fPV>(arrTempPar[19].fTempSet+ABS(arrTempPar[19].fTempArea)) OR arrTempCtrl[19].Tem_fPV<(arrTempPar[19].fTempSet-ABS(arrTempPar[19].fTempArea))) AND NOT P3User2_Par.Oven_Shield[13] AND P3_SystemRUN.iMode=1  THEN
	P3_Tem_Error[19]:=TRUE;//烤箱5的3板温度不在正常设定温度范围内报警
END_IF

IF (arrTempCtrl[20].Tem_fPV>(arrTempPar[20].fTempSet+ABS(arrTempPar[20].fTempArea)) OR arrTempCtrl[20].Tem_fPV<(arrTempPar[20].fTempSet-ABS(arrTempPar[20].fTempArea))) AND NOT P3User2_Par.Oven_Shield[13] AND P3_SystemRUN.iMode=1 THEN
	P3_Tem_Error[20]:=TRUE;//烤箱5的4板温度不在正常设定温度范围内报警
END_IF

//6号烤箱
IF (arrTempCtrl[21].Tem_fPV>(arrTempPar[21].fTempSet+ABS(arrTempPar[21].fTempArea)) OR arrTempCtrl[21].Tem_fPV<(arrTempPar[21].fTempSet-ABS(arrTempPar[21].fTempArea))) AND NOT P3User2_Par.Oven_Shield[16] AND P3_SystemRUN.iMode=1  THEN
	P3_Tem_Error[21]:=TRUE;//烤箱6的1板温度不在正常设定温度范围内报警
END_IF

IF (arrTempCtrl[22].Tem_fPV>(arrTempPar[22].fTempSet+ABS(arrTempPar[22].fTempArea)) OR arrTempCtrl[22].Tem_fPV<(arrTempPar[22].fTempSet-ABS(arrTempPar[22].fTempArea))) AND NOT P3User2_Par.Oven_Shield[16] AND P3_SystemRUN.iMode=1 THEN
	P3_Tem_Error[22]:=TRUE;//烤箱6的2板温度不在正常设定温度范围内报警
END_IF

IF (arrTempCtrl[23].Tem_fPV>(arrTempPar[23].fTempSet+ABS(arrTempPar[23].fTempArea)) OR arrTempCtrl[23].Tem_fPV<(arrTempPar[23].fTempSet-ABS(arrTempPar[23].fTempArea))) AND NOT P3User2_Par.Oven_Shield[16] AND P3_SystemRUN.iMode=1  THEN
	P3_Tem_Error[23]:=TRUE;//烤箱6的3板温度不在正常设定温度范围内报警
END_IF

IF (arrTempCtrl[24].Tem_fPV>(arrTempPar[24].fTempSet+ABS(arrTempPar[24].fTempArea)) OR arrTempCtrl[24].Tem_fPV<(arrTempPar[24].fTempSet-ABS(arrTempPar[24].fTempArea))) AND NOT P3User2_Par.Oven_Shield[16] AND P3_SystemRUN.iMode=1 THEN
	P3_Tem_Error[24]:=TRUE;//烤箱6的4板温度不在正常设定温度范围内报警
END_IF

//7号烤箱
IF (arrTempCtrl[25].Tem_fPV>(arrTempPar[25].fTempSet+ABS(arrTempPar[25].fTempArea)) OR arrTempCtrl[25].Tem_fPV<(arrTempPar[25].fTempSet-ABS(arrTempPar[25].fTempArea))) AND NOT P3User2_Par.Oven_Shield[19] AND P3_SystemRUN.iMode=1  THEN
	P3_Tem_Error[25]:=TRUE;//烤箱7的1板温度不在正常设定温度范围内报警
END_IF

IF (arrTempCtrl[26].Tem_fPV>(arrTempPar[26].fTempSet+ABS(arrTempPar[26].fTempArea)) OR arrTempCtrl[26].Tem_fPV<(arrTempPar[26].fTempSet-ABS(arrTempPar[26].fTempArea))) AND NOT P3User2_Par.Oven_Shield[19] AND P3_SystemRUN.iMode=1 THEN
	P3_Tem_Error[26]:=TRUE;//烤箱7的2板温度不在正常设定温度范围内报警
END_IF

IF (arrTempCtrl[27].Tem_fPV>(arrTempPar[27].fTempSet+ABS(arrTempPar[27].fTempArea)) OR arrTempCtrl[27].Tem_fPV<(arrTempPar[27].fTempSet-ABS(arrTempPar[27].fTempArea))) AND NOT P3User2_Par.Oven_Shield[19] AND P3_SystemRUN.iMode=1  THEN
	P3_Tem_Error[27]:=TRUE;//烤箱7的3板温度不在正常设定温度范围内报警
END_IF

IF (arrTempCtrl[28].Tem_fPV>(arrTempPar[28].fTempSet+ABS(arrTempPar[28].fTempArea)) OR arrTempCtrl[28].Tem_fPV<(arrTempPar[28].fTempSet-ABS(arrTempPar[28].fTempArea))) AND NOT P3User2_Par.Oven_Shield[19] AND P3_SystemRUN.iMode=1 THEN
	P3_Tem_Error[28]:=TRUE;//烤箱7的4板温度不在正常设定温度范围内报警
END_IF

//8号烤箱
IF (arrTempCtrl[33].Tem_fPV>(arrTempPar[33].fTempSet+ABS(arrTempPar[33].fTempArea)) OR arrTempCtrl[33].Tem_fPV<(arrTempPar[33].fTempSet-ABS(arrTempPar[33].fTempArea))) AND NOT P3User2_Par.Oven_Shield[2] AND P3_SystemRUN.iMode=1  THEN
	P3_Tem_Error[33]:=TRUE;//烤箱8的1板温度不在正常设定温度范围内报警
END_IF

IF (arrTempCtrl[34].Tem_fPV>(arrTempPar[34].fTempSet+ABS(arrTempPar[34].fTempArea)) OR arrTempCtrl[34].Tem_fPV<(arrTempPar[34].fTempSet-ABS(arrTempPar[34].fTempArea))) AND NOT P3User2_Par.Oven_Shield[2] AND P3_SystemRUN.iMode=1 THEN
	P3_Tem_Error[34]:=TRUE;//烤箱8的2板温度不在正常设定温度范围内报警
END_IF

IF (arrTempCtrl[35].Tem_fPV>(arrTempPar[35].fTempSet+ABS(arrTempPar[35].fTempArea)) OR arrTempCtrl[35].Tem_fPV<(arrTempPar[35].fTempSet-ABS(arrTempPar[35].fTempArea))) AND NOT P3User2_Par.Oven_Shield[2] AND P3_SystemRUN.iMode=1  THEN
	P3_Tem_Error[35]:=TRUE;//烤箱8的3板温度不在正常设定温度范围内报警
END_IF

IF (arrTempCtrl[36].Tem_fPV>(arrTempPar[36].fTempSet+ABS(arrTempPar[36].fTempArea)) OR arrTempCtrl[36].Tem_fPV<(arrTempPar[36].fTempSet-ABS(arrTempPar[36].fTempArea))) AND NOT P3User2_Par.Oven_Shield[2] AND P3_SystemRUN.iMode=1 THEN
	P3_Tem_Error[36]:=TRUE;//烤箱8的4板温度不在正常设定温度范围内报警
END_IF

//9号烤箱
IF (arrTempCtrl[37].Tem_fPV>(arrTempPar[37].fTempSet+ABS(arrTempPar[37].fTempArea)) OR arrTempCtrl[37].Tem_fPV<(arrTempPar[37].fTempSet-ABS(arrTempPar[37].fTempArea))) AND NOT P3User2_Par.Oven_Shield[5] AND P3_SystemRUN.iMode=1  THEN
	P3_Tem_Error[37]:=TRUE;//烤箱9的1板温度不在正常设定温度范围内报警
END_IF

IF (arrTempCtrl[38].Tem_fPV>(arrTempPar[38].fTempSet+ABS(arrTempPar[38].fTempArea)) OR arrTempCtrl[38].Tem_fPV<(arrTempPar[38].fTempSet-ABS(arrTempPar[38].fTempArea))) AND NOT P3User2_Par.Oven_Shield[5] AND P3_SystemRUN.iMode=1 THEN
	P3_Tem_Error[38]:=TRUE;//烤箱9的2板温度不在正常设定温度范围内报警
END_IF

IF (arrTempCtrl[39].Tem_fPV>(arrTempPar[39].fTempSet+ABS(arrTempPar[39].fTempArea)) OR arrTempCtrl[39].Tem_fPV<(arrTempPar[39].fTempSet-ABS(arrTempPar[39].fTempArea))) AND NOT P3User2_Par.Oven_Shield[5] AND P3_SystemRUN.iMode=1  THEN
	P3_Tem_Error[39]:=TRUE;//烤箱9的3板温度不在正常设定温度范围内报警
END_IF

IF (arrTempCtrl[40].Tem_fPV>(arrTempPar[40].fTempSet+ABS(arrTempPar[40].fTempArea)) OR arrTempCtrl[40].Tem_fPV<(arrTempPar[40].fTempSet-ABS(arrTempPar[40].fTempArea))) AND NOT P3User2_Par.Oven_Shield[5] AND P3_SystemRUN.iMode=1 THEN
	P3_Tem_Error[40]:=TRUE;//烤箱9的4板温度不在正常设定温度范围内报警
END_IF

//10号烤箱
IF (arrTempCtrl[41].Tem_fPV>(arrTempPar[41].fTempSet+ABS(arrTempPar[41].fTempArea)) OR arrTempCtrl[41].Tem_fPV<(arrTempPar[41].fTempSet-ABS(arrTempPar[41].fTempArea))) AND NOT P3User2_Par.Oven_Shield[8] AND P3_SystemRUN.iMode=1  THEN
	P3_Tem_Error[41]:=TRUE;//烤箱10的1板温度不在正常设定温度范围内报警
END_IF

IF (arrTempCtrl[42].Tem_fPV>(arrTempPar[42].fTempSet+ABS(arrTempPar[42].fTempArea)) OR arrTempCtrl[42].Tem_fPV<(arrTempPar[42].fTempSet-ABS(arrTempPar[42].fTempArea))) AND NOT P3User2_Par.Oven_Shield[8] AND P3_SystemRUN.iMode=1 THEN
	P3_Tem_Error[42]:=TRUE;//烤箱10的2板温度不在正常设定温度范围内报警
END_IF

IF (arrTempCtrl[43].Tem_fPV>(arrTempPar[43].fTempSet+ABS(arrTempPar[43].fTempArea)) OR arrTempCtrl[43].Tem_fPV<(arrTempPar[43].fTempSet-ABS(arrTempPar[43].fTempArea))) AND NOT P3User2_Par.Oven_Shield[8] AND P3_SystemRUN.iMode=1  THEN
	P3_Tem_Error[43]:=TRUE;//烤箱10的3板温度不在正常设定温度范围内报警
END_IF

IF (arrTempCtrl[44].Tem_fPV>(arrTempPar[44].fTempSet+ABS(arrTempPar[44].fTempArea)) OR arrTempCtrl[44].Tem_fPV<(arrTempPar[44].fTempSet-ABS(arrTempPar[44].fTempArea))) AND NOT P3User2_Par.Oven_Shield[8] AND P3_SystemRUN.iMode=1 THEN
	P3_Tem_Error[44]:=TRUE;//烤箱10的4板温度不在正常设定温度范围内报警
END_IF

//11号烤箱
IF (arrTempCtrl[45].Tem_fPV>(arrTempPar[45].fTempSet+ABS(arrTempPar[45].fTempArea)) OR arrTempCtrl[45].Tem_fPV<(arrTempPar[45].fTempSet-ABS(arrTempPar[45].fTempArea))) AND NOT P3User2_Par.Oven_Shield[11] AND P3_SystemRUN.iMode=1  THEN
	P3_Tem_Error[45]:=TRUE;//烤箱11的1板温度不在正常设定温度范围内报警
END_IF

IF (arrTempCtrl[46].Tem_fPV>(arrTempPar[46].fTempSet+ABS(arrTempPar[46].fTempArea)) OR arrTempCtrl[46].Tem_fPV<(arrTempPar[46].fTempSet-ABS(arrTempPar[46].fTempArea))) AND NOT P3User2_Par.Oven_Shield[11] AND P3_SystemRUN.iMode=1 THEN
	P3_Tem_Error[46]:=TRUE;//烤箱11的2板温度不在正常设定温度范围内报警
END_IF

IF (arrTempCtrl[47].Tem_fPV>(arrTempPar[47].fTempSet+ABS(arrTempPar[47].fTempArea)) OR arrTempCtrl[47].Tem_fPV<(arrTempPar[47].fTempSet-ABS(arrTempPar[47].fTempArea))) AND NOT P3User2_Par.Oven_Shield[11] AND P3_SystemRUN.iMode=1  THEN
	P3_Tem_Error[47]:=TRUE;//烤箱11的3板温度不在正常设定温度范围内报警
END_IF

IF (arrTempCtrl[48].Tem_fPV>(arrTempPar[48].fTempSet+ABS(arrTempPar[48].fTempArea)) OR arrTempCtrl[48].Tem_fPV<(arrTempPar[48].fTempSet-ABS(arrTempPar[48].fTempArea))) AND NOT P3User2_Par.Oven_Shield[11] AND P3_SystemRUN.iMode=1 THEN
	P3_Tem_Error[48]:=TRUE;//烤箱11的4板温度不在正常设定温度范围内报警
END_IF

//12号烤箱
IF (arrTempCtrl[49].Tem_fPV>(arrTempPar[49].fTempSet+ABS(arrTempPar[49].fTempArea)) OR arrTempCtrl[49].Tem_fPV<(arrTempPar[49].fTempSet-ABS(arrTempPar[49].fTempArea))) AND NOT P3User2_Par.Oven_Shield[14] AND P3_SystemRUN.iMode=1  THEN
	P3_Tem_Error[49]:=TRUE;//烤箱12的1板温度不在正常设定温度范围内报警
END_IF

IF (arrTempCtrl[50].Tem_fPV>(arrTempPar[50].fTempSet+ABS(arrTempPar[50].fTempArea)) OR arrTempCtrl[50].Tem_fPV<(arrTempPar[50].fTempSet-ABS(arrTempPar[50].fTempArea))) AND NOT P3User2_Par.Oven_Shield[14] AND P3_SystemRUN.iMode=1 THEN
	P3_Tem_Error[50]:=TRUE;//烤箱12的2板温度不在正常设定温度范围内报警
END_IF

IF (arrTempCtrl[51].Tem_fPV>(arrTempPar[51].fTempSet+ABS(arrTempPar[51].fTempArea)) OR arrTempCtrl[51].Tem_fPV<(arrTempPar[51].fTempSet-ABS(arrTempPar[51].fTempArea))) AND NOT P3User2_Par.Oven_Shield[14] AND P3_SystemRUN.iMode=1  THEN
	P3_Tem_Error[51]:=TRUE;//烤箱12的3板温度不在正常设定温度范围内报警
END_IF

IF (arrTempCtrl[52].Tem_fPV>(arrTempPar[52].fTempSet+ABS(arrTempPar[52].fTempArea)) OR arrTempCtrl[52].Tem_fPV<(arrTempPar[52].fTempSet-ABS(arrTempPar[52].fTempArea))) AND NOT P3User2_Par.Oven_Shield[14] AND P3_SystemRUN.iMode=1 THEN
	P3_Tem_Error[52]:=TRUE;//烤箱12的4板温度不在正常设定温度范围内报警
END_IF

//13号烤箱
IF (arrTempCtrl[53].Tem_fPV>(arrTempPar[53].fTempSet+ABS(arrTempPar[53].fTempArea)) OR arrTempCtrl[53].Tem_fPV<(arrTempPar[53].fTempSet-ABS(arrTempPar[53].fTempArea))) AND NOT P3User2_Par.Oven_Shield[17] AND P3_SystemRUN.iMode=1  THEN
	P3_Tem_Error[53]:=TRUE;//烤箱13的1板温度不在正常设定温度范围内报警
END_IF

IF (arrTempCtrl[54].Tem_fPV>(arrTempPar[54].fTempSet+ABS(arrTempPar[54].fTempArea)) OR arrTempCtrl[54].Tem_fPV<(arrTempPar[54].fTempSet-ABS(arrTempPar[54].fTempArea))) AND NOT P3User2_Par.Oven_Shield[17] AND P3_SystemRUN.iMode=1 THEN
	P3_Tem_Error[54]:=TRUE;//烤箱13的2板温度不在正常设定温度范围内报警
END_IF

IF (arrTempCtrl[55].Tem_fPV>(arrTempPar[55].fTempSet+ABS(arrTempPar[55].fTempArea)) OR arrTempCtrl[55].Tem_fPV<(arrTempPar[55].fTempSet-ABS(arrTempPar[55].fTempArea))) AND NOT P3User2_Par.Oven_Shield[17] AND P3_SystemRUN.iMode=1  THEN
	P3_Tem_Error[55]:=TRUE;//烤箱13的3板温度不在正常设定温度范围内报警
END_IF

IF (arrTempCtrl[56].Tem_fPV>(arrTempPar[56].fTempSet+ABS(arrTempPar[56].fTempArea)) OR arrTempCtrl[56].Tem_fPV<(arrTempPar[56].fTempSet-ABS(arrTempPar[56].fTempArea))) AND NOT P3User2_Par.Oven_Shield[17] AND P3_SystemRUN.iMode=1 THEN
	P3_Tem_Error[56]:=TRUE;//烤箱13的4板温度不在正常设定温度范围内报警
END_IF


//14号烤箱
IF (arrTempCtrl[57].Tem_fPV>(arrTempPar[57].fTempSet+ABS(arrTempPar[57].fTempArea)) OR arrTempCtrl[57].Tem_fPV<(arrTempPar[57].fTempSet-ABS(arrTempPar[57].fTempArea))) AND NOT P3User2_Par.Oven_Shield[20] AND P3_SystemRUN.iMode=1  THEN
	P3_Tem_Error[57]:=TRUE;//烤箱14的1板温度不在正常设定温度范围内报警
END_IF

IF (arrTempCtrl[58].Tem_fPV>(arrTempPar[58].fTempSet+ABS(arrTempPar[58].fTempArea)) OR arrTempCtrl[58].Tem_fPV<(arrTempPar[58].fTempSet-ABS(arrTempPar[58].fTempArea))) AND NOT P3User2_Par.Oven_Shield[20] AND P3_SystemRUN.iMode=1 THEN
	P3_Tem_Error[58]:=TRUE;//烤箱14的2板温度不在正常设定温度范围内报警
END_IF

IF (arrTempCtrl[59].Tem_fPV>(arrTempPar[59].fTempSet+ABS(arrTempPar[59].fTempArea)) OR arrTempCtrl[59].Tem_fPV<(arrTempPar[59].fTempSet-ABS(arrTempPar[59].fTempArea))) AND NOT P3User2_Par.Oven_Shield[20] AND P3_SystemRUN.iMode=1  THEN
	P3_Tem_Error[59]:=TRUE;//烤箱14的3板温度不在正常设定温度范围内报警
END_IF

IF (arrTempCtrl[60].Tem_fPV>(arrTempPar[60].fTempSet+ABS(arrTempPar[60].fTempArea)) OR arrTempCtrl[60].Tem_fPV<(arrTempPar[60].fTempSet-ABS(arrTempPar[60].fTempArea))) AND NOT P3User2_Par.Oven_Shield[20] AND P3_SystemRUN.iMode=1 THEN
	P3_Tem_Error[60]:=TRUE;//烤箱14的4板温度不在正常设定温度范围内报警
END_IF




//15号烤箱
IF (arrTempCtrl[65].Tem_fPV>(arrTempPar[65].fTempSet+ABS(arrTempPar[65].fTempArea)) OR arrTempCtrl[65].Tem_fPV<(arrTempPar[65].fTempSet-ABS(arrTempPar[65].fTempArea))) AND NOT P3User2_Par.Oven_Shield[3] AND P3_SystemRUN.iMode=1  THEN
	P3_Tem_Error[65]:=TRUE;//烤箱15的1板温度不在正常设定温度范围内报警
END_IF

IF (arrTempCtrl[66].Tem_fPV>(arrTempPar[66].fTempSet+ABS(arrTempPar[66].fTempArea)) OR arrTempCtrl[66].Tem_fPV<(arrTempPar[66].fTempSet-ABS(arrTempPar[66].fTempArea))) AND NOT P3User2_Par.Oven_Shield[3] AND P3_SystemRUN.iMode=1 THEN
	P3_Tem_Error[66]:=TRUE;//烤箱15的2板温度不在正常设定温度范围内报警
END_IF

IF (arrTempCtrl[67].Tem_fPV>(arrTempPar[67].fTempSet+ABS(arrTempPar[67].fTempArea)) OR arrTempCtrl[67].Tem_fPV<(arrTempPar[67].fTempSet-ABS(arrTempPar[67].fTempArea))) AND NOT P3User2_Par.Oven_Shield[3] AND P3_SystemRUN.iMode=1  THEN
	P3_Tem_Error[67]:=TRUE;//烤箱15的3板温度不在正常设定温度范围内报警
END_IF

IF (arrTempCtrl[68].Tem_fPV>(arrTempPar[68].fTempSet+ABS(arrTempPar[68].fTempArea)) OR arrTempCtrl[68].Tem_fPV<(arrTempPar[68].fTempSet-ABS(arrTempPar[68].fTempArea))) AND NOT P3User2_Par.Oven_Shield[3] AND P3_SystemRUN.iMode=1 THEN
	P3_Tem_Error[68]:=TRUE;//烤箱15的4板温度不在正常设定温度范围内报警
END_IF


//16号烤箱
IF (arrTempCtrl[69].Tem_fPV>(arrTempPar[69].fTempSet+ABS(arrTempPar[69].fTempArea)) OR arrTempCtrl[69].Tem_fPV<(arrTempPar[69].fTempSet-ABS(arrTempPar[69].fTempArea))) AND NOT P3User2_Par.Oven_Shield[6] AND P3_SystemRUN.iMode=1  THEN
	P3_Tem_Error[69]:=TRUE;//烤箱16的1板温度不在正常设定温度范围内报警
END_IF

IF (arrTempCtrl[70].Tem_fPV>(arrTempPar[70].fTempSet+ABS(arrTempPar[70].fTempArea)) OR arrTempCtrl[70].Tem_fPV<(arrTempPar[70].fTempSet-ABS(arrTempPar[70].fTempArea))) AND NOT P3User2_Par.Oven_Shield[6] AND P3_SystemRUN.iMode=1 THEN
	P3_Tem_Error[70]:=TRUE;//烤箱16的2板温度不在正常设定温度范围内报警
END_IF

IF (arrTempCtrl[71].Tem_fPV>(arrTempPar[71].fTempSet+ABS(arrTempPar[71].fTempArea)) OR arrTempCtrl[71].Tem_fPV<(arrTempPar[71].fTempSet-ABS(arrTempPar[71].fTempArea))) AND NOT P3User2_Par.Oven_Shield[6] AND P3_SystemRUN.iMode=1  THEN
	P3_Tem_Error[71]:=TRUE;//烤箱16的3板温度不在正常设定温度范围内报警
END_IF

IF (arrTempCtrl[72].Tem_fPV>(arrTempPar[72].fTempSet+ABS(arrTempPar[72].fTempArea)) OR arrTempCtrl[72].Tem_fPV<(arrTempPar[72].fTempSet-ABS(arrTempPar[72].fTempArea))) AND NOT P3User2_Par.Oven_Shield[6] AND P3_SystemRUN.iMode=1 THEN
	P3_Tem_Error[72]:=TRUE;//烤箱16的4板温度不在正常设定温度范围内报警
END_IF


//17号烤箱
IF (arrTempCtrl[73].Tem_fPV>(arrTempPar[73].fTempSet+ABS(arrTempPar[73].fTempArea)) OR arrTempCtrl[73].Tem_fPV<(arrTempPar[73].fTempSet-ABS(arrTempPar[73].fTempArea))) AND NOT P3User2_Par.Oven_Shield[9] AND P3_SystemRUN.iMode=1  THEN
	P3_Tem_Error[73]:=TRUE;//烤箱17的1板温度不在正常设定温度范围内报警
END_IF

IF (arrTempCtrl[74].Tem_fPV>(arrTempPar[74].fTempSet+ABS(arrTempPar[74].fTempArea)) OR arrTempCtrl[74].Tem_fPV<(arrTempPar[74].fTempSet-ABS(arrTempPar[74].fTempArea))) AND NOT P3User2_Par.Oven_Shield[9] AND P3_SystemRUN.iMode=1 THEN
	P3_Tem_Error[74]:=TRUE;//烤箱17的2板温度不在正常设定温度范围内报警
END_IF

IF (arrTempCtrl[75].Tem_fPV>(arrTempPar[75].fTempSet+ABS(arrTempPar[75].fTempArea)) OR arrTempCtrl[75].Tem_fPV<(arrTempPar[75].fTempSet-ABS(arrTempPar[75].fTempArea))) AND NOT P3User2_Par.Oven_Shield[9] AND P3_SystemRUN.iMode=1  THEN
	P3_Tem_Error[75]:=TRUE;//烤箱17的3板温度不在正常设定温度范围内报警
END_IF

IF (arrTempCtrl[76].Tem_fPV>(arrTempPar[76].fTempSet+ABS(arrTempPar[76].fTempArea)) OR arrTempCtrl[76].Tem_fPV<(arrTempPar[76].fTempSet-ABS(arrTempPar[76].fTempArea))) AND NOT P3User2_Par.Oven_Shield[9] AND P3_SystemRUN.iMode=1 THEN
	P3_Tem_Error[76]:=TRUE;//烤箱17的4板温度不在正常设定温度范围内报警
END_IF


//18号烤箱
IF (arrTempCtrl[77].Tem_fPV>(arrTempPar[77].fTempSet+ABS(arrTempPar[77].fTempArea)) OR arrTempCtrl[77].Tem_fPV<(arrTempPar[77].fTempSet-ABS(arrTempPar[77].fTempArea))) AND NOT P3User2_Par.Oven_Shield[12] AND P3_SystemRUN.iMode=1  THEN
	P3_Tem_Error[77]:=TRUE;//烤箱18的1板温度不在正常设定温度范围内报警
END_IF

IF (arrTempCtrl[78].Tem_fPV>(arrTempPar[78].fTempSet+ABS(arrTempPar[78].fTempArea)) OR arrTempCtrl[78].Tem_fPV<(arrTempPar[78].fTempSet-ABS(arrTempPar[78].fTempArea))) AND NOT P3User2_Par.Oven_Shield[12] AND P3_SystemRUN.iMode=1 THEN
	P3_Tem_Error[78]:=TRUE;//烤箱18的2板温度不在正常设定温度范围内报警
END_IF

IF (arrTempCtrl[79].Tem_fPV>(arrTempPar[79].fTempSet+ABS(arrTempPar[79].fTempArea)) OR arrTempCtrl[79].Tem_fPV<(arrTempPar[79].fTempSet-ABS(arrTempPar[79].fTempArea))) AND NOT P3User2_Par.Oven_Shield[12] AND P3_SystemRUN.iMode=1  THEN
	P3_Tem_Error[79]:=TRUE;//烤箱18的3板温度不在正常设定温度范围内报警
END_IF

IF (arrTempCtrl[80].Tem_fPV>(arrTempPar[80].fTempSet+ABS(arrTempPar[80].fTempArea)) OR arrTempCtrl[80].Tem_fPV<(arrTempPar[80].fTempSet-ABS(arrTempPar[80].fTempArea))) AND NOT P3User2_Par.Oven_Shield[12] AND P3_SystemRUN.iMode=1 THEN
	P3_Tem_Error[80]:=TRUE;//烤箱18的4板温度不在正常设定温度范围内报警
END_IF


//19号烤箱
IF (arrTempCtrl[81].Tem_fPV>(arrTempPar[81].fTempSet+ABS(arrTempPar[81].fTempArea)) OR arrTempCtrl[81].Tem_fPV<(arrTempPar[81].fTempSet-ABS(arrTempPar[81].fTempArea))) AND NOT P3User2_Par.Oven_Shield[15] AND P3_SystemRUN.iMode=1  THEN
	P3_Tem_Error[81]:=TRUE;//烤箱19的1板温度不在正常设定温度范围内报警
END_IF

IF (arrTempCtrl[82].Tem_fPV>(arrTempPar[82].fTempSet+ABS(arrTempPar[82].fTempArea)) OR arrTempCtrl[82].Tem_fPV<(arrTempPar[82].fTempSet-ABS(arrTempPar[82].fTempArea))) AND NOT P3User2_Par.Oven_Shield[15] AND P3_SystemRUN.iMode=1 THEN
	P3_Tem_Error[82]:=TRUE;//烤箱19的2板温度不在正常设定温度范围内报警
END_IF

IF (arrTempCtrl[83].Tem_fPV>(arrTempPar[83].fTempSet+ABS(arrTempPar[83].fTempArea)) OR arrTempCtrl[83].Tem_fPV<(arrTempPar[83].fTempSet-ABS(arrTempPar[83].fTempArea))) AND NOT P3User2_Par.Oven_Shield[15] AND P3_SystemRUN.iMode=1  THEN
	P3_Tem_Error[83]:=TRUE;//烤箱19的3板温度不在正常设定温度范围内报警
END_IF

IF (arrTempCtrl[84].Tem_fPV>(arrTempPar[84].fTempSet+ABS(arrTempPar[84].fTempArea)) OR arrTempCtrl[84].Tem_fPV<(arrTempPar[84].fTempSet-ABS(arrTempPar[84].fTempArea))) AND NOT P3User2_Par.Oven_Shield[15] AND P3_SystemRUN.iMode=1 THEN
	P3_Tem_Error[84]:=TRUE;//烤箱19的4板温度不在正常设定温度范围内报警
END_IF


//20号烤箱
IF (arrTempCtrl[85].Tem_fPV>(arrTempPar[85].fTempSet+ABS(arrTempPar[85].fTempArea)) OR arrTempCtrl[85].Tem_fPV<(arrTempPar[85].fTempSet-ABS(arrTempPar[85].fTempArea))) AND NOT P3User2_Par.Oven_Shield[18] AND P3_SystemRUN.iMode=1  THEN
	P3_Tem_Error[85]:=TRUE;//烤箱20的1板温度不在正常设定温度范围内报警
END_IF

IF (arrTempCtrl[86].Tem_fPV>(arrTempPar[86].fTempSet+ABS(arrTempPar[86].fTempArea)) OR arrTempCtrl[86].Tem_fPV<(arrTempPar[86].fTempSet-ABS(arrTempPar[86].fTempArea))) AND NOT P3User2_Par.Oven_Shield[18] AND P3_SystemRUN.iMode=1 THEN
	P3_Tem_Error[86]:=TRUE;//烤箱20的2板温度不在正常设定温度范围内报警
END_IF

IF (arrTempCtrl[87].Tem_fPV>(arrTempPar[87].fTempSet+ABS(arrTempPar[87].fTempArea)) OR arrTempCtrl[87].Tem_fPV<(arrTempPar[87].fTempSet-ABS(arrTempPar[87].fTempArea))) AND NOT P3User2_Par.Oven_Shield[18] AND P3_SystemRUN.iMode=1  THEN
	P3_Tem_Error[87]:=TRUE;//烤箱20的3板温度不在正常设定温度范围内报警
END_IF

IF (arrTempCtrl[88].Tem_fPV>(arrTempPar[88].fTempSet+ABS(arrTempPar[88].fTempArea)) OR arrTempCtrl[88].Tem_fPV<(arrTempPar[88].fTempSet-ABS(arrTempPar[88].fTempArea))) AND NOT P3User2_Par.Oven_Shield[18] AND P3_SystemRUN.iMode=1 THEN
	P3_Tem_Error[88]:=TRUE;//烤箱20的4板温度不在正常设定温度范围内报警
END_IF


//21号烤箱
IF (arrTempCtrl[89].Tem_fPV>(arrTempPar[89].fTempSet+ABS(arrTempPar[89].fTempArea)) OR arrTempCtrl[89].Tem_fPV<(arrTempPar[89].fTempSet-ABS(arrTempPar[89].fTempArea))) AND NOT P3User2_Par.Oven_Shield[21] AND P3_SystemRUN.iMode=1  THEN
	P3_Tem_Error[89]:=TRUE;//烤箱21的1板温度不在正常设定温度范围内报警
END_IF

IF (arrTempCtrl[90].Tem_fPV>(arrTempPar[90].fTempSet+ABS(arrTempPar[90].fTempArea)) OR arrTempCtrl[90].Tem_fPV<(arrTempPar[90].fTempSet-ABS(arrTempPar[90].fTempArea))) AND NOT P3User2_Par.Oven_Shield[21] AND P3_SystemRUN.iMode=1 THEN
	P3_Tem_Error[90]:=TRUE;//烤箱21的2板温度不在正常设定温度范围内报警
END_IF

IF (arrTempCtrl[91].Tem_fPV>(arrTempPar[91].fTempSet+ABS(arrTempPar[91].fTempArea)) OR arrTempCtrl[91].Tem_fPV<(arrTempPar[91].fTempSet-ABS(arrTempPar[91].fTempArea))) AND NOT P3User2_Par.Oven_Shield[21] AND P3_SystemRUN.iMode=1  THEN
	P3_Tem_Error[91]:=TRUE;//烤箱21的3板温度不在正常设定温度范围内报警
END_IF

IF (arrTempCtrl[92].Tem_fPV>(arrTempPar[92].fTempSet+ABS(arrTempPar[92].fTempArea)) OR arrTempCtrl[92].Tem_fPV<(arrTempPar[92].fTempSet-ABS(arrTempPar[92].fTempArea))) AND NOT P3User2_Par.Oven_Shield[21] AND P3_SystemRUN.iMode=1 THEN
	P3_Tem_Error[92]:=TRUE;//烤箱21的4板温度不在正常设定温度范围内报警
END_IF




//热压
IF (arrTempCtrl[93].Tem_fPV>(arrTempPar[93].fTempSet+ABS(arrTempPar[93].fTempArea)) OR arrTempCtrl[93].Tem_fPV<(arrTempPar[93].fTempSet-ABS(arrTempPar[93].fTempArea))) AND P3_SystemRUN.iMode=1  THEN
	P3_Tem_Error[93]:=TRUE;//热压上板温度不在正常设定温度范围内报警
END_IF

IF (arrTempCtrl[94].Tem_fPV>(arrTempPar[94].fTempSet+ABS(arrTempPar[94].fTempArea)) OR arrTempCtrl[94].Tem_fPV<(arrTempPar[94].fTempSet-ABS(arrTempPar[94].fTempArea))) AND P3_SystemRUN.iMode=1 THEN
	P3_Tem_Error[94]:=TRUE;//热压下板温度不在正常设定温度范围内报警
END_IF

ACTION ACT2:
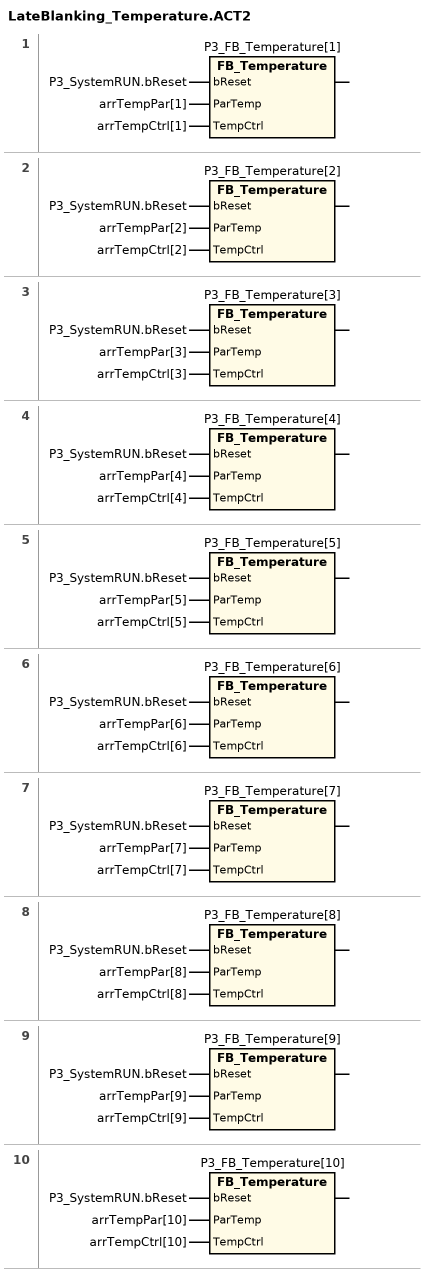
// NETWORK 1
P3_FB_Temperature[1](bReset := P3_SystemRUN.bReset, ParTemp := arrTempPar[1], TempCtrl := arrTempCtrl[1]); // FB_Temperature

// NETWORK 2
P3_FB_Temperature[2](bReset := P3_SystemRUN.bReset, ParTemp := arrTempPar[2], TempCtrl := arrTempCtrl[2]); // FB_Temperature

// NETWORK 3
P3_FB_Temperature[3](bReset := P3_SystemRUN.bReset, ParTemp := arrTempPar[3], TempCtrl := arrTempCtrl[3]); // FB_Temperature

// NETWORK 4
P3_FB_Temperature[4](bReset := P3_SystemRUN.bReset, ParTemp := arrTempPar[4], TempCtrl := arrTempCtrl[4]); // FB_Temperature

// NETWORK 5
P3_FB_Temperature[5](bReset := P3_SystemRUN.bReset, ParTemp := arrTempPar[5], TempCtrl := arrTempCtrl[5]); // FB_Temperature

// NETWORK 6
P3_FB_Temperature[6](bReset := P3_SystemRUN.bReset, ParTemp := arrTempPar[6], TempCtrl := arrTempCtrl[6]); // FB_Temperature

// NETWORK 7
P3_FB_Temperature[7](bReset := P3_SystemRUN.bReset, ParTemp := arrTempPar[7], TempCtrl := arrTempCtrl[7]); // FB_Temperature

// NETWORK 8
P3_FB_Temperature[8](bReset := P3_SystemRUN.bReset, ParTemp := arrTempPar[8], TempCtrl := arrTempCtrl[8]); // FB_Temperature

// NETWORK 9
P3_FB_Temperature[9](bReset := P3_SystemRUN.bReset, ParTemp := arrTempPar[9], TempCtrl := arrTempCtrl[9]); // FB_Temperature

// NETWORK 10
P3_FB_Temperature[10](bReset := P3_SystemRUN.bReset, ParTemp := arrTempPar[10], TempCtrl := arrTempCtrl[10]); // FB_Temperature

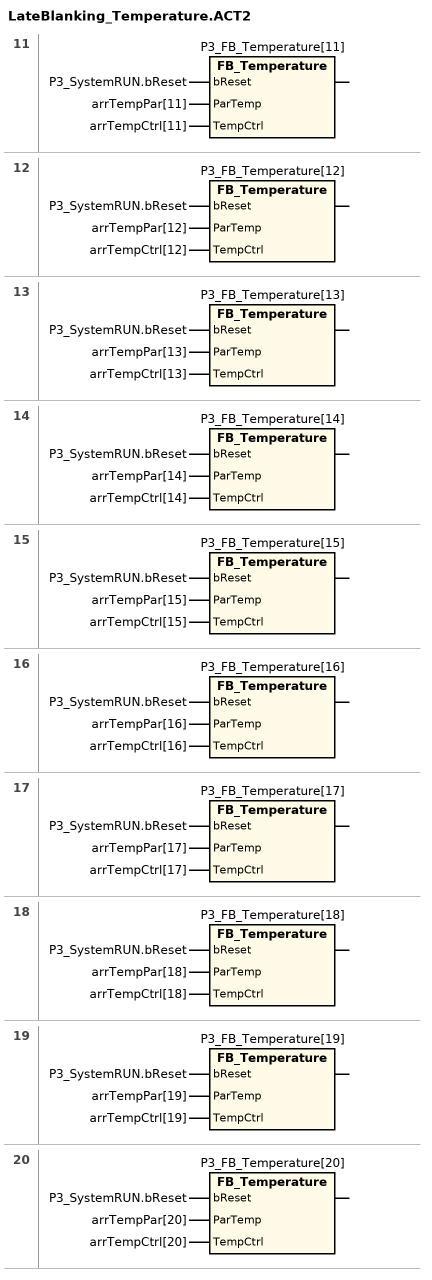
// NETWORK 11
P3_FB_Temperature[11](bReset := P3_SystemRUN.bReset, ParTemp := arrTempPar[11], TempCtrl := arrTempCtrl[11]); // FB_Temperature

// NETWORK 12
P3_FB_Temperature[12](bReset := P3_SystemRUN.bReset, ParTemp := arrTempPar[12], TempCtrl := arrTempCtrl[12]); // FB_Temperature

// NETWORK 13
P3_FB_Temperature[13](bReset := P3_SystemRUN.bReset, ParTemp := arrTempPar[13], TempCtrl := arrTempCtrl[13]); // FB_Temperature

// NETWORK 14
P3_FB_Temperature[14](bReset := P3_SystemRUN.bReset, ParTemp := arrTempPar[14], TempCtrl := arrTempCtrl[14]); // FB_Temperature

// NETWORK 15
P3_FB_Temperature[15](bReset := P3_SystemRUN.bReset, ParTemp := arrTempPar[15], TempCtrl := arrTempCtrl[15]); // FB_Temperature

// NETWORK 16
P3_FB_Temperature[16](bReset := P3_SystemRUN.bReset, ParTemp := arrTempPar[16], TempCtrl := arrTempCtrl[16]); // FB_Temperature

// NETWORK 17
P3_FB_Temperature[17](bReset := P3_SystemRUN.bReset, ParTemp := arrTempPar[17], TempCtrl := arrTempCtrl[17]); // FB_Temperature

// NETWORK 18
P3_FB_Temperature[18](bReset := P3_SystemRUN.bReset, ParTemp := arrTempPar[18], TempCtrl := arrTempCtrl[18]); // FB_Temperature

// NETWORK 19
P3_FB_Temperature[19](bReset := P3_SystemRUN.bReset, ParTemp := arrTempPar[19], TempCtrl := arrTempCtrl[19]); // FB_Temperature

// NETWORK 20
P3_FB_Temperature[20](bReset := P3_SystemRUN.bReset, ParTemp := arrTempPar[20], TempCtrl := arrTempCtrl[20]); // FB_Temperature

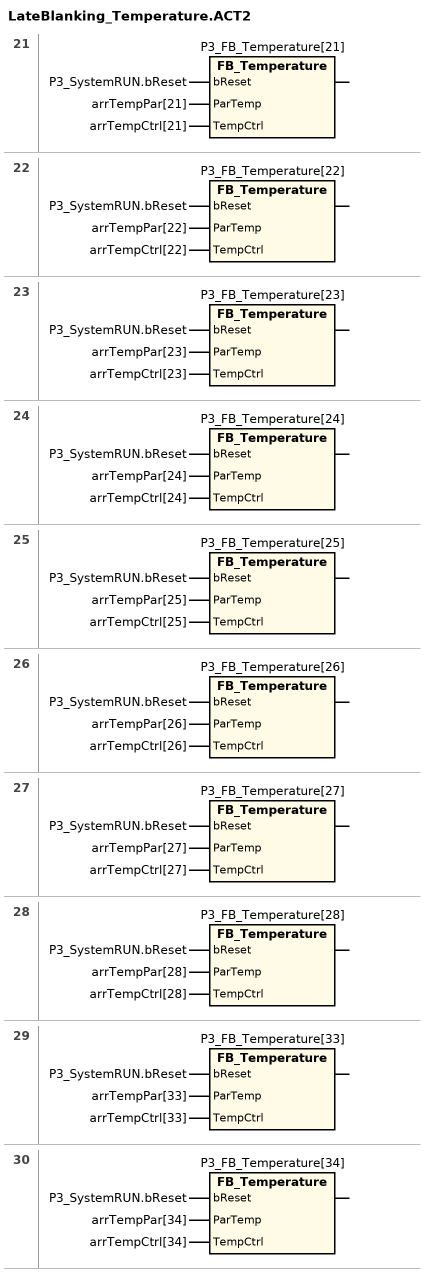
// NETWORK 21
P3_FB_Temperature[21](bReset := P3_SystemRUN.bReset, ParTemp := arrTempPar[21], TempCtrl := arrTempCtrl[21]); // FB_Temperature

// NETWORK 22
P3_FB_Temperature[22](bReset := P3_SystemRUN.bReset, ParTemp := arrTempPar[22], TempCtrl := arrTempCtrl[22]); // FB_Temperature

// NETWORK 23
P3_FB_Temperature[23](bReset := P3_SystemRUN.bReset, ParTemp := arrTempPar[23], TempCtrl := arrTempCtrl[23]); // FB_Temperature

// NETWORK 24
P3_FB_Temperature[24](bReset := P3_SystemRUN.bReset, ParTemp := arrTempPar[24], TempCtrl := arrTempCtrl[24]); // FB_Temperature

// NETWORK 25
P3_FB_Temperature[25](bReset := P3_SystemRUN.bReset, ParTemp := arrTempPar[25], TempCtrl := arrTempCtrl[25]); // FB_Temperature

// NETWORK 26
P3_FB_Temperature[26](bReset := P3_SystemRUN.bReset, ParTemp := arrTempPar[26], TempCtrl := arrTempCtrl[26]); // FB_Temperature

// NETWORK 27
P3_FB_Temperature[27](bReset := P3_SystemRUN.bReset, ParTemp := arrTempPar[27], TempCtrl := arrTempCtrl[27]); // FB_Temperature

// NETWORK 28
P3_FB_Temperature[28](bReset := P3_SystemRUN.bReset, ParTemp := arrTempPar[28], TempCtrl := arrTempCtrl[28]); // FB_Temperature

// NETWORK 29
P3_FB_Temperature[33](bReset := P3_SystemRUN.bReset, ParTemp := arrTempPar[33], TempCtrl := arrTempCtrl[33]); // FB_Temperature

// NETWORK 30
P3_FB_Temperature[34](bReset := P3_SystemRUN.bReset, ParTemp := arrTempPar[34], TempCtrl := arrTempCtrl[34]); // FB_Temperature

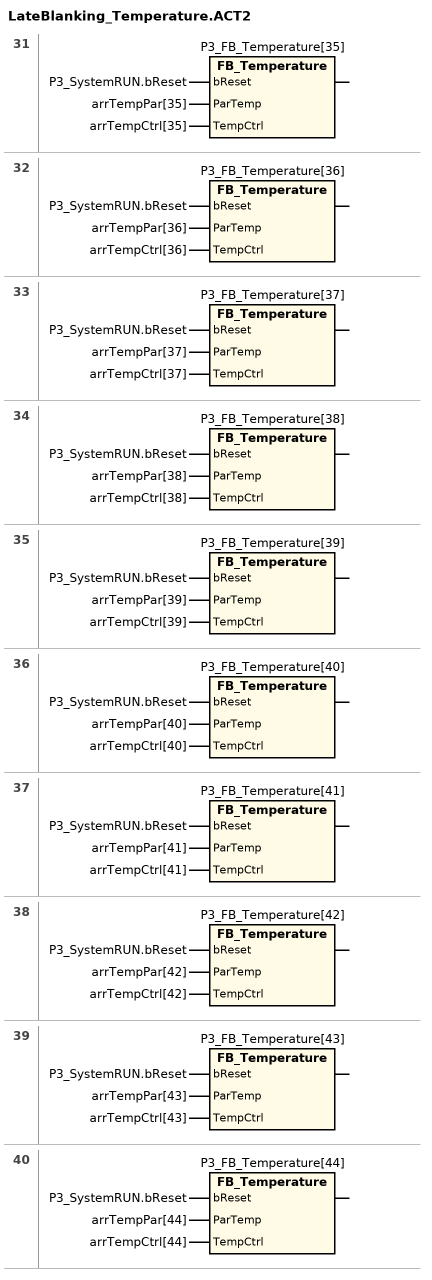
// NETWORK 31
P3_FB_Temperature[35](bReset := P3_SystemRUN.bReset, ParTemp := arrTempPar[35], TempCtrl := arrTempCtrl[35]); // FB_Temperature

// NETWORK 32
P3_FB_Temperature[36](bReset := P3_SystemRUN.bReset, ParTemp := arrTempPar[36], TempCtrl := arrTempCtrl[36]); // FB_Temperature

// NETWORK 33
P3_FB_Temperature[37](bReset := P3_SystemRUN.bReset, ParTemp := arrTempPar[37], TempCtrl := arrTempCtrl[37]); // FB_Temperature

// NETWORK 34
P3_FB_Temperature[38](bReset := P3_SystemRUN.bReset, ParTemp := arrTempPar[38], TempCtrl := arrTempCtrl[38]); // FB_Temperature

// NETWORK 35
P3_FB_Temperature[39](bReset := P3_SystemRUN.bReset, ParTemp := arrTempPar[39], TempCtrl := arrTempCtrl[39]); // FB_Temperature

// NETWORK 36
P3_FB_Temperature[40](bReset := P3_SystemRUN.bReset, ParTemp := arrTempPar[40], TempCtrl := arrTempCtrl[40]); // FB_Temperature

// NETWORK 37
P3_FB_Temperature[41](bReset := P3_SystemRUN.bReset, ParTemp := arrTempPar[41], TempCtrl := arrTempCtrl[41]); // FB_Temperature

// NETWORK 38
P3_FB_Temperature[42](bReset := P3_SystemRUN.bReset, ParTemp := arrTempPar[42], TempCtrl := arrTempCtrl[42]); // FB_Temperature

// NETWORK 39
P3_FB_Temperature[43](bReset := P3_SystemRUN.bReset, ParTemp := arrTempPar[43], TempCtrl := arrTempCtrl[43]); // FB_Temperature

// NETWORK 40
P3_FB_Temperature[44](bReset := P3_SystemRUN.bReset, ParTemp := arrTempPar[44], TempCtrl := arrTempCtrl[44]); // FB_Temperature

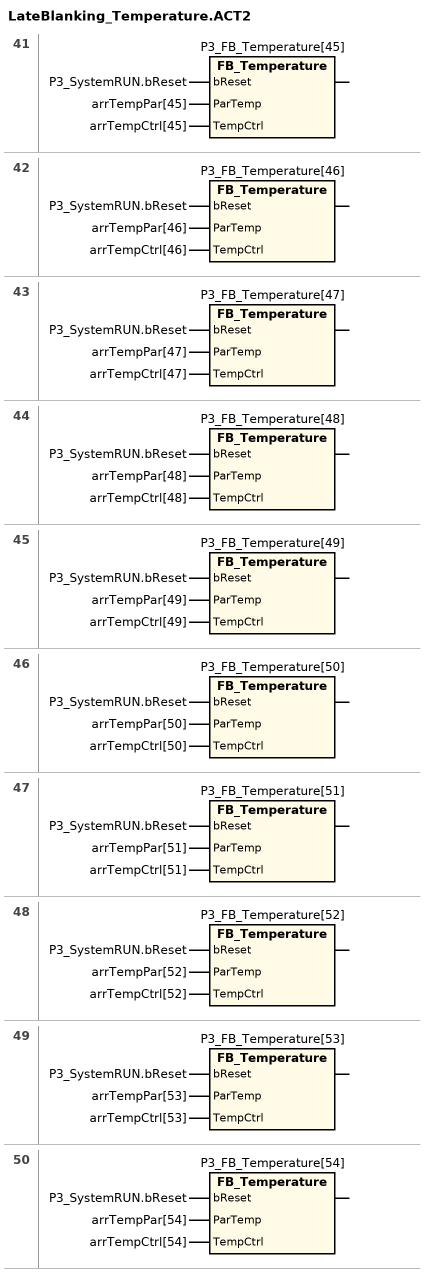
// NETWORK 41
P3_FB_Temperature[45](bReset := P3_SystemRUN.bReset, ParTemp := arrTempPar[45], TempCtrl := arrTempCtrl[45]); // FB_Temperature

// NETWORK 42
P3_FB_Temperature[46](bReset := P3_SystemRUN.bReset, ParTemp := arrTempPar[46], TempCtrl := arrTempCtrl[46]); // FB_Temperature

// NETWORK 43
P3_FB_Temperature[47](bReset := P3_SystemRUN.bReset, ParTemp := arrTempPar[47], TempCtrl := arrTempCtrl[47]); // FB_Temperature

// NETWORK 44
P3_FB_Temperature[48](bReset := P3_SystemRUN.bReset, ParTemp := arrTempPar[48], TempCtrl := arrTempCtrl[48]); // FB_Temperature

// NETWORK 45
P3_FB_Temperature[49](bReset := P3_SystemRUN.bReset, ParTemp := arrTempPar[49], TempCtrl := arrTempCtrl[49]); // FB_Temperature

// NETWORK 46
P3_FB_Temperature[50](bReset := P3_SystemRUN.bReset, ParTemp := arrTempPar[50], TempCtrl := arrTempCtrl[50]); // FB_Temperature

// NETWORK 47
P3_FB_Temperature[51](bReset := P3_SystemRUN.bReset, ParTemp := arrTempPar[51], TempCtrl := arrTempCtrl[51]); // FB_Temperature

// NETWORK 48
P3_FB_Temperature[52](bReset := P3_SystemRUN.bReset, ParTemp := arrTempPar[52], TempCtrl := arrTempCtrl[52]); // FB_Temperature

// NETWORK 49
P3_FB_Temperature[53](bReset := P3_SystemRUN.bReset, ParTemp := arrTempPar[53], TempCtrl := arrTempCtrl[53]); // FB_Temperature

// NETWORK 50
P3_FB_Temperature[54](bReset := P3_SystemRUN.bReset, ParTemp := arrTempPar[54], TempCtrl := arrTempCtrl[54]); // FB_Temperature

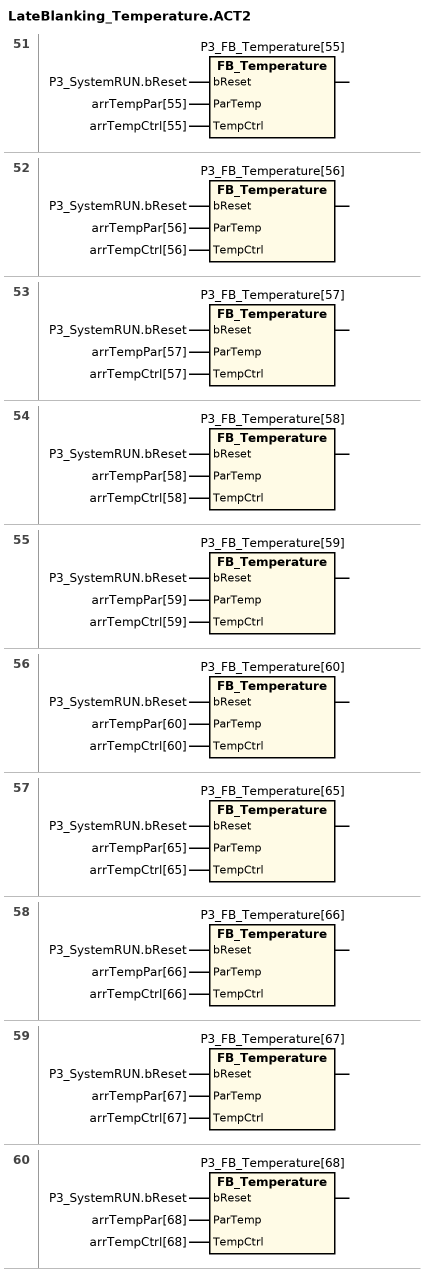
// NETWORK 51
P3_FB_Temperature[55](bReset := P3_SystemRUN.bReset, ParTemp := arrTempPar[55], TempCtrl := arrTempCtrl[55]); // FB_Temperature

// NETWORK 52
P3_FB_Temperature[56](bReset := P3_SystemRUN.bReset, ParTemp := arrTempPar[56], TempCtrl := arrTempCtrl[56]); // FB_Temperature

// NETWORK 53
P3_FB_Temperature[57](bReset := P3_SystemRUN.bReset, ParTemp := arrTempPar[57], TempCtrl := arrTempCtrl[57]); // FB_Temperature

// NETWORK 54
P3_FB_Temperature[58](bReset := P3_SystemRUN.bReset, ParTemp := arrTempPar[58], TempCtrl := arrTempCtrl[58]); // FB_Temperature

// NETWORK 55
P3_FB_Temperature[59](bReset := P3_SystemRUN.bReset, ParTemp := arrTempPar[59], TempCtrl := arrTempCtrl[59]); // FB_Temperature

// NETWORK 56
P3_FB_Temperature[60](bReset := P3_SystemRUN.bReset, ParTemp := arrTempPar[60], TempCtrl := arrTempCtrl[60]); // FB_Temperature

// NETWORK 57
P3_FB_Temperature[65](bReset := P3_SystemRUN.bReset, ParTemp := arrTempPar[65], TempCtrl := arrTempCtrl[65]); // FB_Temperature

// NETWORK 58
P3_FB_Temperature[66](bReset := P3_SystemRUN.bReset, ParTemp := arrTempPar[66], TempCtrl := arrTempCtrl[66]); // FB_Temperature

// NETWORK 59
P3_FB_Temperature[67](bReset := P3_SystemRUN.bReset, ParTemp := arrTempPar[67], TempCtrl := arrTempCtrl[67]); // FB_Temperature

// NETWORK 60
P3_FB_Temperature[68](bReset := P3_SystemRUN.bReset, ParTemp := arrTempPar[68], TempCtrl := arrTempCtrl[68]); // FB_Temperature

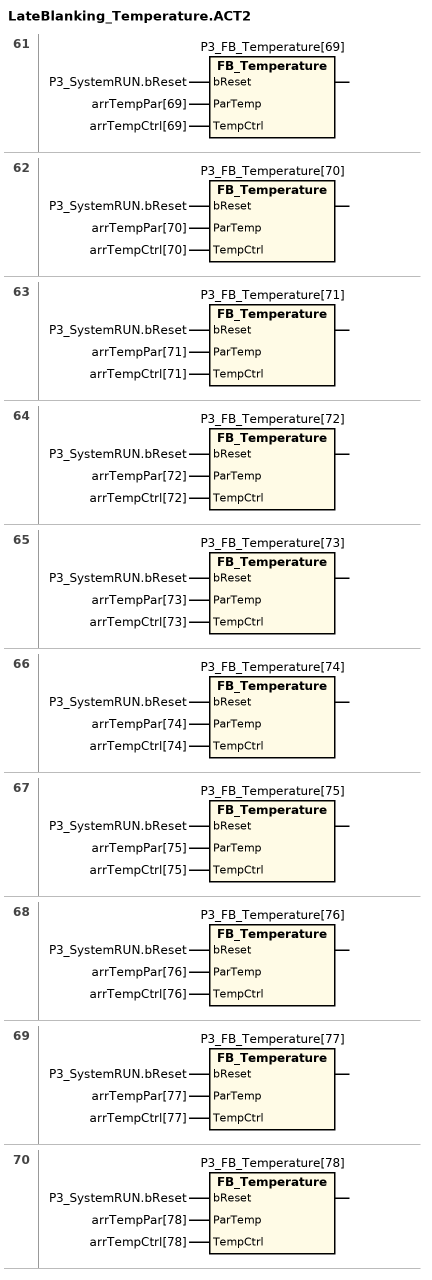
// NETWORK 61
P3_FB_Temperature[69](bReset := P3_SystemRUN.bReset, ParTemp := arrTempPar[69], TempCtrl := arrTempCtrl[69]); // FB_Temperature

// NETWORK 62
P3_FB_Temperature[70](bReset := P3_SystemRUN.bReset, ParTemp := arrTempPar[70], TempCtrl := arrTempCtrl[70]); // FB_Temperature

// NETWORK 63
P3_FB_Temperature[71](bReset := P3_SystemRUN.bReset, ParTemp := arrTempPar[71], TempCtrl := arrTempCtrl[71]); // FB_Temperature

// NETWORK 64
P3_FB_Temperature[72](bReset := P3_SystemRUN.bReset, ParTemp := arrTempPar[72], TempCtrl := arrTempCtrl[72]); // FB_Temperature

// NETWORK 65
P3_FB_Temperature[73](bReset := P3_SystemRUN.bReset, ParTemp := arrTempPar[73], TempCtrl := arrTempCtrl[73]); // FB_Temperature

// NETWORK 66
P3_FB_Temperature[74](bReset := P3_SystemRUN.bReset, ParTemp := arrTempPar[74], TempCtrl := arrTempCtrl[74]); // FB_Temperature

// NETWORK 67
P3_FB_Temperature[75](bReset := P3_SystemRUN.bReset, ParTemp := arrTempPar[75], TempCtrl := arrTempCtrl[75]); // FB_Temperature

// NETWORK 68
P3_FB_Temperature[76](bReset := P3_SystemRUN.bReset, ParTemp := arrTempPar[76], TempCtrl := arrTempCtrl[76]); // FB_Temperature

// NETWORK 69
P3_FB_Temperature[77](bReset := P3_SystemRUN.bReset, ParTemp := arrTempPar[77], TempCtrl := arrTempCtrl[77]); // FB_Temperature

